LIN {X 0,Y 139.748,Z 528.406,A -85,B 0,C 180,E1 -25612.878,E2 -25612.878} C_VEL
LIN {X 0,Y 135.039,Z 532.973,A -85,B 0,C 180,E1 -25616.378,E2 -25616.378} C_VEL
LIN {X 0,Y 130.036,Z 537.238,A -85,B 0,C 180,E1 -25620.892,E2 -25620.892} C_VEL
LIN {X 0,Y 125.044,Z 540.854,A -85,B 0,C 180,E1 -25626.83,E2 -25626.83} C_VEL
LIN {X 0,Y 123.078,Z 542.06,A -85,B 0,C 180,E1 -25629.962,E2 -25629.962} C_VEL
LIN {X 0,Y 120.547,Z 543.249,A -85,B 0,C 180,E1 -25636.512,E2 -25636.512} C_VEL
LIN {X 0,Y 119.471,Z 542.937,A -85,B 0,C 180,E1 -25643.241,E2 -25643.241} C_VEL
LIN {X 0,Y 119.487,Z 541.317,A -85,B 0,C 180,E1 -25649.219,E2 -25649.219} C_VEL
LIN {X 0,Y 119.402,Z 538.391,A -85,B 0,C 180,E1 -25655.063,E2 -25655.063} C_VEL
LIN {X 0,Y 119.834,Z 534.742,A -85,B 0,C 180,E1 -25660.131,E2 -25660.131} C_VEL
LIN {X 0,Y 120.849,Z 529.936,A -85,B 0,C 180,E1 -25665.168,E2 -25665.168} C_VEL
LIN {X 0,Y 122.779,Z 523.85,A -85,B 0,C 180,E1 -25670.084,E2 -25670.084} C_VEL
LIN {X 0,Y 125.465,Z 516.248,A -85,B 0,C 180,E1 -25674.839,E2 -25674.839} C_VEL
LIN {X 0,Y 127.649,Z 509.707,A -85,B 0,C 180,E1 -25678.109,E2 -25678.109} C_VEL
LIN {X 0,Y 129.2,Z 505.909,A -85,B 0,C 180,E1 -25679.699,E2 -25679.699} C_VEL
LIN {X 0,Y 130.221,Z 501.642,A -85,B 0,C 180,E1 -25681.43,E2 -25681.43} C_VEL
LIN {X 0,Y 130.169,Z 494.346,A -85,B 0,C 180,E1 -25684.371,E2 -25684.371} C_VEL
LIN {X 0,Y 130.081,Z 486.628,A -85,B 0,C 180,E1 -25687.131,E2 -25687.131} C_VEL
LIN {X 0,Y 130.988,Z 481.594,A -85,B 0,C 180,E1 -25688.495,E2 -25688.495} C_VEL
LIN {X 0,Y 133.452,Z 473.066,A -85,B 0,C 180,E1 -25690.171,E2 -25690.171} C_VEL
LIN {X 0,Y 136.354,Z 460.646,A -85,B 0,C 180,E1 -25692.067,E2 -25692.067} C_VEL
LIN {X 0,Y 138.723,Z 447.504,A -85,B 0,C 180,E1 -25693.398,E2 -25693.398} C_VEL
LIN {X 0,Y 140.113,Z 434.838,A -85,B 0,C 180,E1 -25694.224,E2 -25694.224} C_VEL
LIN {X 0,Y 142.429,Z 397.329,A -85,B 0,C 180,E1 -25695.919,E2 -25695.919} C_VEL
LIN {X 0,Y 141.717,Z 386.256,A -85,B 0,C 180,E1 -25696.887,E2 -25696.887} C_VEL
LIN {X 0,Y 137.465,Z 373.788,A -85,B 0,C 180,E1 -25699.297,E2 -25699.297} C_VEL
LIN {X 0,Y 132.823,Z 362.78,A -85,B 0,C 180,E1 -25702.028,E2 -25702.028} C_VEL
LIN {X 0,Y 127.538,Z 354.274,A -85,B 0,C 180,E1 -25705.197,E2 -25705.197} C_VEL
LIN {X 0,Y 124.389,Z 349.812,A -85,B 0,C 180,E1 -25707.263,E2 -25707.263} C_VEL
LIN {X 0,Y 121.952,Z 346.24,A -85,B 0,C 180,E1 -25709.016,E2 -25709.016} C_VEL
LIN {X 0,Y 119.65,Z 343.536,A -85,B 0,C 180,E1 -25710.739,E2 -25710.739} C_VEL
LIN {X 0,Y 118.548,Z 341.533,A -85,B 0,C 180,E1 -25711.688,E2 -25711.688} C_VEL
LIN {X 0,Y 116.07,Z 339.331,A -85,B 0,C 180,E1 -25713.719,E2 -25713.719} C_VEL
LIN {X 0,Y 114.968,Z 336.772,A -85,B 0,C 180,E1 -25714.875,E2 -25714.875} C_VEL
LIN {X 0,Y 114.899,Z 336.166,A -85,B 0,C 180,E1 -25715.068,E2 -25715.068} C_VEL
LIN {X 0,Y 114.974,Z 336.161,A -85,B 0,C 180,E1 -25718.484,E2 -25718.484} C_VEL
LIN {X 0,Y 115.14,Z 336.126,A -85,B 0,C 180,E1 -25725.868,E2 -25725.868} C_VEL
LIN {X 0,Y 115.38,Z 336.107,A -85,B 0,C 180,E1 -25729.471,E2 -25729.471} C_VEL
LIN {X 0,Y 115.524,Z 336.065,A -85,B 0,C 180,E1 -25736.512,E2 -25736.512} C_VEL
LIN {X 0,Y 115.985,Z 336.035,A -85,B 0,C 180,E1 -25740,E2 -25740} C_VEL
LIN {X 0,Y 115.35,Z 336.07,A -85,B 0,C 180,E1 -25746.999,E2 -25746.999} C_VEL
LIN {X 0,Y 115.242,Z 336.129,A -85,B 0,C 180,E1 -25752.658,E2 -25752.658} C_VEL
LIN {X 0,Y 115.003,Z 336.158,A -85,B 0,C 180,E1 -25757.792,E2 -25757.792} C_VEL
LIN {X 0,Y 114.94,Z 336.162,A -85,B 0,C 180,E1 -25763.492,E2 -25763.492} C_VEL
LIN {X 0,Y 114.857,Z 336.175,A -85,B 0,C 180,E1 -25771.064,E2 -25771.064} C_VEL
LIN {X 0,Y 114.77,Z 336.18,A -85,B 0,C 180,E1 -25777.76,E2 -25777.76} C_VEL
LIN {X 0,Y 114.826,Z 336.337,A -85,B 0,C 180,E1 -25779.563,E2 -25779.563} C_VEL
LIN {X 0,Y 115.753,Z 338.963,A -85,B 0,C 180,E1 -25780.602,E2 -25780.602} C_VEL
LIN {X 0,Y 117.898,Z 341.218,A -85,B 0,C 180,E1 -25782.432,E2 -25782.432} C_VEL
LIN {X 0,Y 118.746,Z 341.779,A -85,B 0,C 180,E1 -25783.08,E2 -25783.08} C_VEL
LIN {X 0,Y 120.61,Z 344.977,A -85,B 0,C 180,E1 -25784.635,E2 -25784.635} C_VEL
LIN {X 0,Y 122.547,Z 347.185,A -85,B 0,C 180,E1 -25786.04,E2 -25786.04} C_VEL
LIN {X 0,Y 125.082,Z 350.706,A -85,B 0,C 180,E1 -25787.81,E2 -25787.81} C_VEL
LIN {X 0,Y 130.98,Z 359.656,A -85,B 0,C 180,E1 -25791.51,E2 -25791.51} C_VEL
LIN {X 0,Y 135.931,Z 368.292,A -85,B 0,C 180,E1 -25794.301,E2 -25794.301} C_VEL
LIN {X 0,Y 140.566,Z 377.554,A -85,B 0,C 180,E1 -25796.725,E2 -25796.725} C_VEL
LIN {X 0,Y 143.321,Z 384.36,A -85,B 0,C 180,E1 -25798.137,E2 -25798.137} C_VEL
LIN {X 0,Y 139.982,Z 431.241,A -85,B 0,C 180,E1 -25800.18,E2 -25800.18} C_VEL
LIN {X 0,Y 138.259,Z 444.693,A -85,B 0,C 180,E1 -25801.285,E2 -25801.285} C_VEL
LIN {X 0,Y 135.688,Z 457.591,A -85,B 0,C 180,E1 -25802.845,E2 -25802.845} C_VEL
LIN {X 0,Y 132.84,Z 469.466,A -85,B 0,C 180,E1 -25804.963,E2 -25804.963} C_VEL
LIN {X 0,Y 129.653,Z 480.844,A -85,B 0,C 180,E1 -25807.704,E2 -25807.704} C_VEL
LIN {X 0,Y 126.054,Z 491.183,A -85,B 0,C 180,E1 -25810.882,E2 -25810.882} C_VEL
LIN {X 0,Y 122.214,Z 501.266,A -85,B 0,C 180,E1 -25815.005,E2 -25815.005} C_VEL
LIN {X 0,Y 118.712,Z 510.135,A -85,B 0,C 180,E1 -25819.772,E2 -25819.772} C_VEL
LIN {X 0,Y 115.976,Z 517.221,A -85,B 0,C 180,E1 -25824.787,E2 -25824.787} C_VEL
LIN {X 0,Y 114.01,Z 522.883,A -85,B 0,C 180,E1 -25830.003,E2 -25830.003} C_VEL
LIN {X 0,Y 112.849,Z 526.966,A -85,B 0,C 180,E1 -25834.827,E2 -25834.827} C_VEL
LIN {X 0,Y 111.978,Z 530.745,A -85,B 0,C 180,E1 -25840.855,E2 -25840.855} C_VEL
LIN {X 0,Y 111.907,Z 532.439,A -85,B 0,C 180,E1 -25844.552,E2 -25844.552} C_VEL
LIN {X 0,Y 112.52,Z 534.256,A -85,B 0,C 180,E1 -25850.461,E2 -25850.461} C_VEL
LIN {X 0,Y 113.757,Z 534.966,A -85,B 0,C 180,E1 -25855.627,E2 -25855.627} C_VEL
LIN {X 0,Y 116.732,Z 534.61,A -85,B 0,C 180,E1 -25862.553,E2 -25862.553} C_VEL
LIN {X 0,Y 118.978,Z 533.699,A -85,B 0,C 180,E1 -25866.209,E2 -25866.209} C_VEL
LIN {X 0,Y 121.486,Z 532.41,A -85,B 0,C 180,E1 -25869.523,E2 -25869.523} C_VEL
LIN {X 0,Y 125.754,Z 529.728,A -85,B 0,C 180,E1 -25874.093,E2 -25874.093} C_VEL
LIN {X 0,Y 131.124,Z 525.728,A -85,B 0,C 180,E1 -25878.625,E2 -25878.625} C_VEL
LIN {X 0,Y 137.011,Z 520.617,A -85,B 0,C 180,E1 -25882.665,E2 -25882.665} C_VEL
LIN {X 0,Y 143.466,Z 514.096,A -85,B 0,C 180,E1 -25886.388,E2 -25886.388} C_VEL
LIN {X 0,Y 150.547,Z 505.857,A -85,B 0,C 180,E1 -25889.73,E2 -25889.73} C_VEL
LIN {X 0,Y 156.825,Z 497.394,A -85,B 0,C 180,E1 -25892.264,E2 -25892.264} C_VEL
LIN {X 0,Y 162.673,Z 488.098,A -85,B 0,C 180,E1 -25894.403,E2 -25894.403} C_VEL
LIN {X 0,Y 168.006,Z 477.877,A -85,B 0,C 180,E1 -25896.218,E2 -25896.218} C_VEL
LIN {X 0,Y 172.799,Z 466.653,A -85,B 0,C 180,E1 -25897.713,E2 -25897.713} C_VEL
LIN {X 0,Y 176.818,Z 454.72,A -85,B 0,C 180,E1 -25898.887,E2 -25898.887} C_VEL
LIN {X 0,Y 180.007,Z 441.516,A -85,B 0,C 180,E1 -25899.83,E2 -25899.83} C_VEL
LIN {X 0,Y 181.953,Z 429.077,A -85,B 0,C 180,E1 -25900.379,E2 -25900.379} C_VEL
LIN {X 0,Y 183.021,Z 417.526,A -85,B 0,C 180,E1 -25900.768,E2 -25900.768} C_VEL
LIN {X 0,Y 179.727,Z 410.839,A -85,B 0,C 180,E1 -25903.603,E2 -25903.603} C_VEL
LIN {X 0,Y 176.506,Z 404.889,A -85,B 0,C 180,E1 -25906.783,E2 -25906.783} C_VEL
LIN {X 0,Y 174.369,Z 401.21,A -85,B 0,C 180,E1 -25909.226,E2 -25909.226} C_VEL
LIN {X 0,Y 172.892,Z 398.642,A -85,B 0,C 180,E1 -25911.166,E2 -25911.166} C_VEL
LIN {X 0,Y 170.702,Z 394.74,A -85,B 0,C 180,E1 -25914.759,E2 -25914.759} C_VEL
LIN {X 0,Y 168.911,Z 391.63,A -85,B 0,C 180,E1 -25918.878,E2 -25918.878} C_VEL
LIN {X 0,Y 168.596,Z 390.672,A -85,B 0,C 180,E1 -25920,E2 -25920} C_VEL
LIN {X 0,Y 167.449,Z 390.036,A -85,B 0,C 180,E1 -25927.233,E2 -25927.233} C_VEL
LIN {X 0,Y 168.55,Z 391.104,A -85,B 0,C 180,E1 -25933.561,E2 -25933.561} C_VEL
LIN {X 0,Y 170.089,Z 394.454,A -85,B 0,C 180,E1 -25937.726,E2 -25937.726} C_VEL
LIN {X 0,Y 171.264,Z 395.995,A -85,B 0,C 180,E1 -25939.856,E2 -25939.856} C_VEL
LIN {X 0,Y 173.653,Z 401.111,A -85,B 0,C 180,E1 -25943.557,E2 -25943.557} C_VEL
LIN {X 0,Y 175.886,Z 406.084,A -85,B 0,C 180,E1 -25946.348,E2 -25946.348} C_VEL
LIN {X 0,Y 178.896,Z 413.432,A -85,B 0,C 180,E1 -25949.584,E2 -25949.584} C_VEL
LIN {X 0,Y 181.73,Z 420.904,A -85,B 0,C 180,E1 -25952.25,E2 -25952.25} C_VEL
LIN {X 0,Y 182.632,Z 423.59,A -85,B 0,C 180,E1 -25953.058,E2 -25953.058} C_VEL
LIN {X 0,Y 180.595,Z 441.612,A -85,B 0,C 180,E1 -25953.634,E2 -25953.634} C_VEL
LIN {X 0,Y 178.032,Z 454.239,A -85,B 0,C 180,E1 -25954.299,E2 -25954.299} C_VEL
LIN {X 0,Y 174.696,Z 465.563,A -85,B 0,C 180,E1 -25955.135,E2 -25955.135} C_VEL
LIN {X 0,Y 170.087,Z 477.416,A -85,B 0,C 180,E1 -25956.316,E2 -25956.316} C_VEL
LIN {X 0,Y 164.689,Z 488.641,A -85,B 0,C 180,E1 -25957.861,E2 -25957.861} C_VEL
LIN {X 0,Y 159.45,Z 497.74,A -85,B 0,C 180,E1 -25959.524,E2 -25959.524} C_VEL
LIN {X 0,Y 153.164,Z 507.117,A -85,B 0,C 180,E1 -25961.784,E2 -25961.784} C_VEL
LIN {X 0,Y 145.967,Z 516.189,A -85,B 0,C 180,E1 -25964.749,E2 -25964.749} C_VEL
LIN {X 0,Y 139.287,Z 523.526,A -85,B 0,C 180,E1 -25968.042,E2 -25968.042} C_VEL
LIN {X 0,Y 132.255,Z 530.304,A -85,B 0,C 180,E1 -25972.328,E2 -25972.328} C_VEL
LIN {X 0,Y 127.018,Z 534.81,A -85,B 0,C 180,E1 -25976.403,E2 -25976.403} C_VEL
LIN {X 0,Y 123.878,Z 537.201,A -85,B 0,C 180,E1 -25979.294,E2 -25979.294} C_VEL
LIN {X 0,Y 118.533,Z 540.744,A -85,B 0,C 180,E1 -25985.476,E2 -25985.476} C_VEL
LIN {X 0,Y 116.411,Z 541.883,A -85,B 0,C 180,E1 -25988.76,E2 -25988.76} C_VEL
LIN {X 0,Y 113.638,Z 543.001,A -85,B 0,C 180,E1 -25995.675,E2 -25995.675} C_VEL
LIN {X 0,Y 112.423,Z 542.605,A -85,B 0,C 180,E1 -26002.815,E2 -26002.815} C_VEL
LIN {X 0,Y 112.336,Z 541.788,A -85,B 0,C 180,E1 -26006.411,E2 -26006.411} C_VEL
LIN {X 0,Y 112.448,Z 540.571,A -85,B 0,C 180,E1 -26009.997,E2 -26009.997} C_VEL
LIN {X 0,Y 112.322,Z 537.896,A -85,B 0,C 180,E1 -26015.383,E2 -26015.383} C_VEL
LIN {X 0,Y 112.808,Z 534.167,A -85,B 0,C 180,E1 -26020.769,E2 -26020.769} C_VEL
LIN {X 0,Y 113.96,Z 529.276,A -85,B 0,C 180,E1 -26026.109,E2 -26026.109} C_VEL
LIN {X 0,Y 116.116,Z 523.102,A -85,B 0,C 180,E1 -26031.291,E2 -26031.291} C_VEL
LIN {X 0,Y 119.034,Z 515.391,A -85,B 0,C 180,E1 -26036.28,E2 -26036.28} C_VEL
LIN {X 0,Y 121.143,Z 509.365,A -85,B 0,C 180,E1 -26039.401,E2 -26039.401} C_VEL
LIN {X 0,Y 124.169,Z 501.883,A -85,B 0,C 180,E1 -26042.524,E2 -26042.524} C_VEL
LIN {X 0,Y 127.226,Z 493.263,A -85,B 0,C 180,E1 -26045.449,E2 -26045.449} C_VEL
LIN {X 0,Y 130.988,Z 481.594,A -85,B 0,C 180,E1 -26048.495,E2 -26048.495} C_VEL
LIN {X 0,Y 132.81,Z 482.641,A -85,B 0,C 180,E1 -26049.896,E2 -26049.896} C_VEL
LIN {X 0,Y 132.81,Z 550.306,A -85,B 0,C 180,E1 -26049.896,E2 -26049.896} C_VEL
LIN {X 0,Y 112.28,Z 550.306,A -85,B 0,C 180,E1 -26012.234,E2 -26012.234} C_VEL
LIN {X 0,Y 112.474,Z 548.306,A -85,B 0,C 180,E1 -26011.219,E2 -26011.219} C_VEL
LIN {X 0,Y 112.474,Z 542.531,A -85,B 0,C 180,E1 -26011.219,E2 -26011.219} C_VEL
LIN {X 0,Y 112.448,Z 540.571,A -85,B 0,C 180,E1 -26009.997,E2 -26009.997} C_VEL
LIN {X 0,Y 111.778,Z 539.247,A -85,B 0,C 180,E1 -26012.914,E2 -26012.914} C_VEL
LIN {X 0,Y 110.234,Z 537.667,A -85,B 0,C 180,E1 -26015.768,E2 -26015.768} C_VEL
LIN {X 0,Y 106.956,Z 533.701,A -85,B 0,C 180,E1 -26021.511,E2 -26021.511} C_VEL
LIN {X 0,Y 106.44,Z 531.242,A -85,B 0,C 180,E1 -26024.43,E2 -26024.43} C_VEL
LIN {X 0,Y 106.591,Z 530.347,A -85,B 0,C 180,E1 -26025.386,E2 -26025.386} C_VEL
LIN {X 0,Y 109.011,Z 523.481,A -85,B 0,C 180,E1 -26031.756,E2 -26031.756} C_VEL
LIN {X 0,Y 112.044,Z 515.913,A -85,B 0,C 180,E1 -26037.046,E2 -26037.046} C_VEL
LIN {X 0,Y 114.579,Z 509.293,A -85,B 0,C 180,E1 -26040.708,E2 -26040.708} C_VEL
LIN {X 0,Y 118.166,Z 500.763,A -85,B 0,C 180,E1 -26044.4,E2 -26044.4} C_VEL
LIN {X 0,Y 121.948,Z 490.799,A -85,B 0,C 180,E1 -26047.755,E2 -26047.755} C_VEL
LIN {X 0,Y 125.592,Z 479.732,A -85,B 0,C 180,E1 -26050.577,E2 -26050.577} C_VEL
LIN {X 0,Y 129.109,Z 467.328,A -85,B 0,C 180,E1 -26052.873,E2 -26052.873} C_VEL
LIN {X 0,Y 131.659,Z 455.809,A -85,B 0,C 180,E1 -26054.422,E2 -26054.422} C_VEL
LIN {X 0,Y 133.704,Z 442.907,A -85,B 0,C 180,E1 -26055.605,E2 -26055.605} C_VEL
LIN {X 0,Y 135.239,Z 426.246,A -85,B 0,C 180,E1 -26056.456,E2 -26056.456} C_VEL
LIN {X 0,Y 136.997,Z 398.059,A -85,B 0,C 180,E1 -26057.77,E2 -26057.77} C_VEL
LIN {X 0,Y 136.479,Z 388.679,A -85,B 0,C 180,E1 -26058.621,E2 -26058.621} C_VEL
LIN {X 0,Y 132.52,Z 376.805,A -85,B 0,C 180,E1 -26061.089,E2 -26061.089} C_VEL
LIN {X 0,Y 128.542,Z 367.126,A -85,B 0,C 180,E1 -26063.638,E2 -26063.638} C_VEL
LIN {X 0,Y 123.671,Z 359.17,A -85,B 0,C 180,E1 -26066.816,E2 -26066.816} C_VEL
LIN {X 0,Y 120.424,Z 354.422,A -85,B 0,C 180,E1 -26069.158,E2 -26069.158} C_VEL
LIN {X 0,Y 118.719,Z 351.939,A -85,B 0,C 180,E1 -26070.492,E2 -26070.492} C_VEL
LIN {X 0,Y 116.153,Z 348.364,A -85,B 0,C 180,E1 -26072.647,E2 -26072.647} C_VEL
LIN {X 0,Y 115.403,Z 347.379,A -85,B 0,C 180,E1 -26073.312,E2 -26073.312} C_VEL
LIN {X 0,Y 113.004,Z 344.653,A -85,B 0,C 180,E1 -26075.533,E2 -26075.533} C_VEL
LIN {X 0,Y 112.136,Z 342.754,A -85,B 0,C 180,E1 -26076.513,E2 -26076.513} C_VEL
LIN {X 0,Y 109.351,Z 340.534,A -85,B 0,C 180,E1 -26079.422,E2 -26079.422} C_VEL
LIN {X 0,Y 108.146,Z 338.142,A -85,B 0,C 180,E1 -26081.039,E2 -26081.039} C_VEL
LIN {X 0,Y 107.916,Z 337.008,A -85,B 0,C 180,E1 -26081.489,E2 -26081.489} C_VEL
LIN {X 0,Y 108.295,Z 336.993,A -85,B 0,C 180,E1 -26088.774,E2 -26088.774} C_VEL
LIN {X 0,Y 108.449,Z 336.942,A -85,B 0,C 180,E1 -26096.285,E2 -26096.285} C_VEL
LIN {X 0,Y 108.934,Z 336.914,A -85,B 0,C 180,E1 -26100,E2 -26100} C_VEL
LIN {X 0,Y 108.29,Z 336.95,A -85,B 0,C 180,E1 -26107.458,E2 -26107.458} C_VEL
LIN {X 0,Y 108.164,Z 337.01,A -85,B 0,C 180,E1 -26112.948,E2 -26112.948} C_VEL
LIN {X 0,Y 107.896,Z 337.045,A -85,B 0,C 180,E1 -26119.007,E2 -26119.007} C_VEL
LIN {X 0,Y 107.853,Z 337.048,A -85,B 0,C 180,E1 -26124.186,E2 -26124.186} C_VEL
LIN {X 0,Y 107.779,Z 337.051,A -85,B 0,C 180,E1 -26132.044,E2 -26132.044} C_VEL
LIN {X 0,Y 107.791,Z 337.079,A -85,B 0,C 180,E1 -26133.001,E2 -26133.001} C_VEL
LIN {X 0,Y 108.532,Z 339.574,A -85,B 0,C 180,E1 -26134.185,E2 -26134.185} C_VEL
LIN {X 0,Y 110.337,Z 341.748,A -85,B 0,C 180,E1 -26136.308,E2 -26136.308} C_VEL
LIN {X 0,Y 112.136,Z 342.983,A -85,B 0,C 180,E1 -26138.119,E2 -26138.119} C_VEL
LIN {X 0,Y 113.99,Z 346.133,A -85,B 0,C 180,E1 -26140.055,E2 -26140.055} C_VEL
LIN {X 0,Y 116.076,Z 348.325,A -85,B 0,C 180,E1 -26141.899,E2 -26141.899} C_VEL
LIN {X 0,Y 118.507,Z 351.77,A -85,B 0,C 180,E1 -26143.957,E2 -26143.957} C_VEL
LIN {X 0,Y 122.71,Z 357.834,A -85,B 0,C 180,E1 -26147.129,E2 -26147.129} C_VEL
LIN {X 0,Y 127.287,Z 364.909,A -85,B 0,C 180,E1 -26150.178,E2 -26150.178} C_VEL
LIN {X 0,Y 132.107,Z 373.666,A -85,B 0,C 180,E1 -26153.097,E2 -26153.097} C_VEL
LIN {X 0,Y 136.401,Z 382.721,A -85,B 0,C 180,E1 -26155.527,E2 -26155.527} C_VEL
LIN {X 0,Y 137.681,Z 385.763,A -85,B 0,C 180,E1 -26156.23,E2 -26156.23} C_VEL
LIN {X 0,Y 137.196,Z 395.421,A -85,B 0,C 180,E1 -26156.722,E2 -26156.722} C_VEL
LIN {X 0,Y 134.337,Z 432.384,A -85,B 0,C 180,E1 -26158.383,E2 -26158.383} C_VEL
LIN {X 0,Y 132.557,Z 445.663,A -85,B 0,C 180,E1 -26159.539,E2 -26159.539} C_VEL
LIN {X 0,Y 129.892,Z 458.101,A -85,B 0,C 180,E1 -26161.084,E2 -26161.084} C_VEL
LIN {X 0,Y 126.9,Z 469.914,A -85,B 0,C 180,E1 -26163.261,E2 -26163.261} C_VEL
LIN {X 0,Y 123.519,Z 481.262,A -85,B 0,C 180,E1 -26166.087,E2 -26166.087} C_VEL
LIN {X 0,Y 119.758,Z 491.562,A -85,B 0,C 180,E1 -26169.386,E2 -26169.386} C_VEL
LIN {X 0,Y 116.017,Z 500.807,A -85,B 0,C 180,E1 -26173.28,E2 -26173.28} C_VEL
LIN {X 0,Y 112.25,Z 509.795,A -85,B 0,C 180,E1 -26178.262,E2 -26178.262} C_VEL
LIN {X 0,Y 109.289,Z 517.025,A -85,B 0,C 180,E1 -26183.541,E2 -26183.541} C_VEL
LIN {X 0,Y 107.457,Z 521.902,A -85,B 0,C 180,E1 -26188.129,E2 -26188.129} C_VEL
LIN {X 0,Y 105.766,Z 527.24,A -85,B 0,C 180,E1 -26194.63,E2 -26194.63} C_VEL
LIN {X 0,Y 104.832,Z 531.272,A -85,B 0,C 180,E1 -26201.605,E2 -26201.605} C_VEL
LIN {X 0,Y 104.865,Z 532.919,A -85,B 0,C 180,E1 -26205.553,E2 -26205.553} C_VEL
LIN {X 0,Y 105.515,Z 534.496,A -85,B 0,C 180,E1 -26211.171,E2 -26211.171} C_VEL
LIN {X 0,Y 107.143,Z 535.263,A -85,B 0,C 180,E1 -26217.336,E2 -26217.336} C_VEL
LIN {X 0,Y 110.164,Z 534.899,A -85,B 0,C 180,E1 -26223.967,E2 -26223.967} C_VEL
LIN {X 0,Y 113.055,Z 533.81,A -85,B 0,C 180,E1 -26228.439,E2 -26228.439} C_VEL
LIN {X 0,Y 118.442,Z 531.011,A -85,B 0,C 180,E1 -26234.598,E2 -26234.598} C_VEL
LIN {X 0,Y 124.371,Z 527.048,A -85,B 0,C 180,E1 -26239.72,E2 -26239.72} C_VEL
LIN {X 0,Y 130.465,Z 522.234,A -85,B 0,C 180,E1 -26243.907,E2 -26243.907} C_VEL
LIN {X 0,Y 137.153,Z 516.07,A -85,B 0,C 180,E1 -26247.728,E2 -26247.728} C_VEL
LIN {X 0,Y 144.434,Z 508.335,A -85,B 0,C 180,E1 -26251.149,E2 -26251.149} C_VEL
LIN {X 0,Y 150.868,Z 500.349,A -85,B 0,C 180,E1 -26253.735,E2 -26253.735} C_VEL
LIN {X 0,Y 157.981,Z 489.84,A -85,B 0,C 180,E1 -26256.246,E2 -26256.246} C_VEL
LIN {X 0,Y 163.765,Z 479.448,A -85,B 0,C 180,E1 -26258.134,E2 -26258.134} C_VEL
LIN {X 0,Y 168.707,Z 468.624,A -85,B 0,C 180,E1 -26259.607,E2 -26259.607} C_VEL
LIN {X 0,Y 172.942,Z 456.896,A -85,B 0,C 180,E1 -26260.775,E2 -26260.775} C_VEL
LIN {X 0,Y 176.438,Z 443.601,A -85,B 0,C 180,E1 -26261.757,E2 -26261.757} C_VEL
LIN {X 0,Y 178.686,Z 430.514,A -85,B 0,C 180,E1 -26262.362,E2 -26262.362} C_VEL
LIN {X 0,Y 179.624,Z 421.086,A -85,B 0,C 180,E1 -26262.683,E2 -26262.683} C_VEL
LIN {X 0,Y 176.362,Z 414.445,A -85,B 0,C 180,E1 -26265.826,E2 -26265.826} C_VEL
LIN {X 0,Y 173.363,Z 408.708,A -85,B 0,C 180,E1 -26269.248,E2 -26269.248} C_VEL
LIN {X 0,Y 171.495,Z 405.334,A -85,B 0,C 180,E1 -26271.797,E2 -26271.797} C_VEL
LIN {X 0,Y 169.432,Z 401.474,A -85,B 0,C 180,E1 -26275.417,E2 -26275.417} C_VEL
LIN {X 0,Y 167.748,Z 398.172,A -85,B 0,C 180,E1 -26279.738,E2 -26279.738} C_VEL
LIN {X 0,Y 167.522,Z 397.584,A -85,B 0,C 180,E1 -26280.601,E2 -26280.601} C_VEL
LIN {X 0,Y 166.614,Z 397.162,A -85,B 0,C 180,E1 -26288.186,E2 -26288.186} C_VEL
LIN {X 0,Y 167.511,Z 398.024,A -85,B 0,C 180,E1 -26293.069,E2 -26293.069} C_VEL
LIN {X 0,Y 169.009,Z 401.381,A -85,B 0,C 180,E1 -26297.378,E2 -26297.378} C_VEL
LIN {X 0,Y 169.972,Z 402.756,A -85,B 0,C 180,E1 -26299.234,E2 -26299.234} C_VEL
LIN {X 0,Y 172.118,Z 407.711,A -85,B 0,C 180,E1 -26302.824,E2 -26302.824} C_VEL
LIN {X 0,Y 174.425,Z 413.222,A -85,B 0,C 180,E1 -26305.883,E2 -26305.883} C_VEL
LIN {X 0,Y 177.479,Z 421.435,A -85,B 0,C 180,E1 -26309.336,E2 -26309.336} C_VEL
LIN {X 0,Y 179.239,Z 426.623,A -85,B 0,C 180,E1 -26311.116,E2 -26311.116} C_VEL
LIN {X 0,Y 177.391,Z 441.802,A -85,B 0,C 180,E1 -26311.609,E2 -26311.609} C_VEL
LIN {X 0,Y 174.597,Z 454.82,A -85,B 0,C 180,E1 -26312.293,E2 -26312.293} C_VEL
LIN {X 0,Y 170.842,Z 466.79,A -85,B 0,C 180,E1 -26313.169,E2 -26313.169} C_VEL
LIN {X 0,Y 166.005,Z 478.585,A -85,B 0,C 180,E1 -26314.354,E2 -26314.354} C_VEL
LIN {X 0,Y 160.443,Z 489.534,A -85,B 0,C 180,E1 -26315.866,E2 -26315.866} C_VEL
LIN {X 0,Y 155.06,Z 498.434,A -85,B 0,C 180,E1 -26317.515,E2 -26317.515} C_VEL
LIN {X 0,Y 148.539,Z 507.598,A -85,B 0,C 180,E1 -26319.747,E2 -26319.747} C_VEL
LIN {X 0,Y 141.079,Z 516.535,A -85,B 0,C 180,E1 -26322.709,E2 -26322.709} C_VEL
LIN {X 0,Y 134.106,Z 523.756,A -85,B 0,C 180,E1 -26326.02,E2 -26326.02} C_VEL
LIN {X 0,Y 128.707,Z 528.661,A -85,B 0,C 180,E1 -26329.059,E2 -26329.059} C_VEL
LIN {X 0,Y 122.463,Z 533.813,A -85,B 0,C 180,E1 -26333.46,E2 -26333.46} C_VEL
LIN {X 0,Y 117.826,Z 537.165,A -85,B 0,C 180,E1 -26337.53,E2 -26337.53} C_VEL
LIN {X 0,Y 114.738,Z 539.1,A -85,B 0,C 180,E1 -26340.655,E2 -26340.655} C_VEL
LIN {X 0,Y 112.099,Z 540.618,A -85,B 0,C 180,E1 -26343.966,E2 -26343.966} C_VEL
LIN {X 0,Y 108.047,Z 542.414,A -85,B 0,C 180,E1 -26351.018,E2 -26351.018} C_VEL
LIN {X 0,Y 105.849,Z 542.713,A -85,B 0,C 180,E1 -26358.508,E2 -26358.508} C_VEL
LIN {X 0,Y 105.36,Z 542.254,A -85,B 0,C 180,E1 -26362.331,E2 -26362.331} C_VEL
LIN {X 0,Y 105.246,Z 541.402,A -85,B 0,C 180,E1 -26366.168,E2 -26366.168} C_VEL
LIN {X 0,Y 105.361,Z 540.151,A -85,B 0,C 180,E1 -26369.997,E2 -26369.997} C_VEL
LIN {X 0,Y 105.244,Z 537.401,A -85,B 0,C 180,E1 -26375.746,E2 -26375.746} C_VEL
LIN {X 0,Y 105.815,Z 533.594,A -85,B 0,C 180,E1 -26381.49,E2 -26381.49} C_VEL
LIN {X 0,Y 106.591,Z 530.347,A -85,B 0,C 180,E1 -26385.386,E2 -26385.386} C_VEL
LIN {X 0,Y 106.842,Z 527.656,A -85,B 0,C 180,E1 -26388.182,E2 -26388.182} C_VEL
LIN {X 0,Y 106.071,Z 522.69,A -85,B 0,C 180,E1 -26392.788,E2 -26392.788} C_VEL
LIN {X 0,Y 105.641,Z 517.186,A -85,B 0,C 180,E1 -26397.269,E2 -26397.269} C_VEL
LIN {X 0,Y 106.395,Z 513.493,A -85,B 0,C 180,E1 -26399.752,E2 -26399.752} C_VEL
LIN {X 0,Y 108.363,Z 508.665,A -85,B 0,C 180,E1 -26402.453,E2 -26402.453} C_VEL
LIN {X 0,Y 111.525,Z 501.632,A -85,B 0,C 180,E1 -26405.652,E2 -26405.652} C_VEL
LIN {X 0,Y 115.468,Z 491.896,A -85,B 0,C 180,E1 -26409.155,E2 -26409.155} C_VEL
LIN {X 0,Y 119.207,Z 481.207,A -85,B 0,C 180,E1 -26412.112,E2 -26412.112} C_VEL
LIN {X 0,Y 121.806,Z 473.035,A -85,B 0,C 180,E1 -26413.815,E2 -26413.815} C_VEL
LIN {X 0,Y 124.996,Z 460.764,A -85,B 0,C 180,E1 -26415.793,E2 -26415.793} C_VEL
LIN {X 0,Y 127.548,Z 448.089,A -85,B 0,C 180,E1 -26417.164,E2 -26417.164} C_VEL
LIN {X 0,Y 129.147,Z 435.331,A -85,B 0,C 180,E1 -26418.057,E2 -26418.057} C_VEL
LIN {X 0,Y 131.72,Z 398.47,A -85,B 0,C 180,E1 -26419.795,E2 -26419.795} C_VEL
LIN {X 0,Y 131.244,Z 390.736,A -85,B 0,C 180,E1 -26420.576,E2 -26420.576} C_VEL
LIN {X 0,Y 127.689,Z 379.75,A -85,B 0,C 180,E1 -26423.018,E2 -26423.018} C_VEL
LIN {X 0,Y 124.131,Z 371.032,A -85,B 0,C 180,E1 -26425.516,E2 -26425.516} C_VEL
LIN {X 0,Y 118.446,Z 361.655,A -85,B 0,C 180,E1 -26429.688,E2 -26429.688} C_VEL
LIN {X 0,Y 115.291,Z 357.178,A -85,B 0,C 180,E1 -26432.302,E2 -26432.302} C_VEL
LIN {X 0,Y 112.703,Z 353.448,A -85,B 0,C 180,E1 -26434.714,E2 -26434.714} C_VEL
LIN {X 0,Y 110.096,Z 350.013,A -85,B 0,C 180,E1 -26437.406,E2 -26437.406} C_VEL
LIN {X 0,Y 109.317,Z 348.812,A -85,B 0,C 180,E1 -26438.305,E2 -26438.305} C_VEL
LIN {X 0,Y 106.806,Z 346.222,A -85,B 0,C 180,E1 -26441.29,E2 -26441.29} C_VEL
LIN {X 0,Y 105.624,Z 343.699,A -85,B 0,C 180,E1 -26443.076,E2 -26443.076} C_VEL
LIN {X 0,Y 103.193,Z 342.076,A -85,B 0,C 180,E1 -26446.635,E2 -26446.635} C_VEL
LIN {X 0,Y 101.462,Z 339.05,A -85,B 0,C 180,E1 -26450.154,E2 -26450.154} C_VEL
LIN {X 0,Y 101.222,Z 337.846,A -85,B 0,C 180,E1 -26451.013,E2 -26451.013} C_VEL
LIN {X 0,Y 101.857,Z 337.795,A -85,B 0,C 180,E1 -26460,E2 -26460} C_VEL
LIN {X 0,Y 101.23,Z 337.831,A -85,B 0,C 180,E1 -26467.982,E2 -26467.982} C_VEL
LIN {X 0,Y 101.093,Z 337.888,A -85,B 0,C 180,E1 -26473.291,E2 -26473.291} C_VEL
LIN {X 0,Y 100.88,Z 338.047,A -85,B 0,C 180,E1 -26483.072,E2 -26483.072} C_VEL
LIN {X 0,Y 101.512,Z 340.341,A -85,B 0,C 180,E1 -26484.858,E2 -26484.858} C_VEL
LIN {X 0,Y 103.55,Z 342.812,A -85,B 0,C 180,E1 -26488.642,E2 -26488.642} C_VEL
LIN {X 0,Y 105.581,Z 343.963,A -85,B 0,C 180,E1 -26491.524,E2 -26491.524} C_VEL
LIN {X 0,Y 107.071,Z 346.904,A -85,B 0,C 180,E1 -26493.708,E2 -26493.708} C_VEL
LIN {X 0,Y 109.754,Z 349.454,A -85,B 0,C 180,E1 -26496.803,E2 -26496.803} C_VEL
LIN {X 0,Y 111.93,Z 352.756,A -85,B 0,C 180,E1 -26499.167,E2 -26499.167} C_VEL
LIN {X 0,Y 113.428,Z 354.516,A -85,B 0,C 180,E1 -26500.595,E2 -26500.595} C_VEL
LIN {X 0,Y 116.973,Z 359.668,A -85,B 0,C 180,E1 -26503.745,E2 -26503.745} C_VEL
LIN {X 0,Y 121.255,Z 366.209,A -85,B 0,C 180,E1 -26507.068,E2 -26507.068} C_VEL
LIN {X 0,Y 126.12,Z 374.655,A -85,B 0,C 180,E1 -26510.415,E2 -26510.415} C_VEL
LIN {X 0,Y 131.022,Z 384.848,A -85,B 0,C 180,E1 -26513.483,E2 -26513.483} C_VEL
LIN {X 0,Y 132.447,Z 388.258,A -85,B 0,C 180,E1 -26514.343,E2 -26514.343} C_VEL
LIN {X 0,Y 128.984,Z 432.357,A -85,B 0,C 180,E1 -26516.355,E2 -26516.355} C_VEL
LIN {X 0,Y 126.99,Z 446.3,A -85,B 0,C 180,E1 -26517.582,E2 -26517.582} C_VEL
LIN {X 0,Y 124.231,Z 458.603,A -85,B 0,C 180,E1 -26519.161,E2 -26519.161} C_VEL
LIN {X 0,Y 121.083,Z 470.363,A -85,B 0,C 180,E1 -26521.393,E2 -26521.393} C_VEL
LIN {X 0,Y 117.494,Z 481.68,A -85,B 0,C 180,E1 -26524.303,E2 -26524.303} C_VEL
LIN {X 0,Y 113.578,Z 491.848,A -85,B 0,C 180,E1 -26527.686,E2 -26527.686} C_VEL
LIN {X 0,Y 109.223,Z 501.984,A -85,B 0,C 180,E1 -26532.206,E2 -26532.206} C_VEL
LIN {X 0,Y 105.291,Z 510.818,A -85,B 0,C 180,E1 -26537.474,E2 -26537.474} C_VEL
LIN {X 0,Y 102.178,Z 517.868,A -85,B 0,C 180,E1 -26543.09,E2 -26543.09} C_VEL
LIN {X 0,Y 100.291,Z 522.676,A -85,B 0,C 180,E1 -26547.995,E2 -26547.995} C_VEL
LIN {X 0,Y 98.682,Z 527.502,A -85,B 0,C 180,E1 -26554.386,E2 -26554.386} C_VEL
LIN {X 0,Y 97.807,Z 530.868,A -85,B 0,C 180,E1 -26560.352,E2 -26560.352} C_VEL
LIN {X 0,Y 97.836,Z 533.395,A -85,B 0,C 180,E1 -26566.702,E2 -26566.702} C_VEL
LIN {X 0,Y 98.529,Z 534.736,A -85,B 0,C 180,E1 -26571.985,E2 -26571.985} C_VEL
LIN {X 0,Y 100.614,Z 535.562,A -85,B 0,C 180,E1 -26579.275,E2 -26579.275} C_VEL
LIN {X 0,Y 103.635,Z 535.192,A -85,B 0,C 180,E1 -26585.532,E2 -26585.532} C_VEL
LIN {X 0,Y 107.343,Z 533.926,A -85,B 0,C 180,E1 -26590.902,E2 -26590.902} C_VEL
LIN {X 0,Y 112.598,Z 531.372,A -85,B 0,C 180,E1 -26596.639,E2 -26596.639} C_VEL
LIN {X 0,Y 117.664,Z 528.296,A -85,B 0,C 180,E1 -26600.943,E2 -26600.943} C_VEL
LIN {X 0,Y 124.655,Z 523.302,A -85,B 0,C 180,E1 -26605.681,E2 -26605.681} C_VEL
LIN {X 0,Y 132.109,Z 516.871,A -85,B 0,C 180,E1 -26609.826,E2 -26609.826} C_VEL
LIN {X 0,Y 139.595,Z 509.363,A -85,B 0,C 180,E1 -26613.207,E2 -26613.207} C_VEL
LIN {X 0,Y 146.386,Z 501.416,A -85,B 0,C 180,E1 -26615.813,E2 -26615.813} C_VEL
LIN {X 0,Y 153.531,Z 491.463,A -85,B 0,C 180,E1 -26618.229,E2 -26618.229} C_VEL
LIN {X 0,Y 159.725,Z 480.965,A -85,B 0,C 180,E1 -26620.141,E2 -26620.141} C_VEL
LIN {X 0,Y 164.813,Z 470.464,A -85,B 0,C 180,E1 -26621.588,E2 -26621.588} C_VEL
LIN {X 0,Y 169.253,Z 459.046,A -85,B 0,C 180,E1 -26622.758,E2 -26622.758} C_VEL
LIN {X 0,Y 172.954,Z 446.065,A -85,B 0,C 180,E1 -26623.727,E2 -26623.727} C_VEL
LIN {X 0,Y 175.375,Z 433.781,A -85,B 0,C 180,E1 -26624.322,E2 -26624.322} C_VEL
LIN {X 0,Y 176.408,Z 424.896,A -85,B 0,C 180,E1 -26624.664,E2 -26624.664} C_VEL
LIN {X 0,Y 173.345,Z 418.352,A -85,B 0,C 180,E1 -26628.026,E2 -26628.026} C_VEL
LIN {X 0,Y 171.129,Z 414.096,A -85,B 0,C 180,E1 -26630.887,E2 -26630.887} C_VEL
LIN {X 0,Y 169.747,Z 411.396,A -85,B 0,C 180,E1 -26633.049,E2 -26633.049} C_VEL
LIN {X 0,Y 168.151,Z 408.176,A -85,B 0,C 180,E1 -26636.155,E2 -26636.155} C_VEL
LIN {X 0,Y 166.657,Z 404.862,A -85,B 0,C 180,E1 -26640.453,E2 -26640.453} C_VEL
LIN {X 0,Y 166.172,Z 404.32,A -85,B 0,C 180,E1 -26642.424,E2 -26642.424} C_VEL
LIN {X 0,Y 165.74,Z 404.194,A -85,B 0,C 180,E1 -26648.229,E2 -26648.229} C_VEL
LIN {X 0,Y 166.523,Z 405.107,A -85,B 0,C 180,E1 -26652.761,E2 -26652.761} C_VEL
LIN {X 0,Y 168.076,Z 408.537,A -85,B 0,C 180,E1 -26657.333,E2 -26657.333} C_VEL
LIN {X 0,Y 168.695,Z 409.559,A -85,B 0,C 180,E1 -26658.6,E2 -26658.6} C_VEL
LIN {X 0,Y 170.61,Z 414.328,A -85,B 0,C 180,E1 -26662.079,E2 -26662.079} C_VEL
LIN {X 0,Y 172.791,Z 420.11,A -85,B 0,C 180,E1 -26665.201,E2 -26665.201} C_VEL
LIN {X 0,Y 175.596,Z 428.284,A -85,B 0,C 180,E1 -26668.596,E2 -26668.596} C_VEL
LIN {X 0,Y 176.04,Z 429.715,A -85,B 0,C 180,E1 -26669.094,E2 -26669.094} C_VEL
LIN {X 0,Y 174.163,Z 443.412,A -85,B 0,C 180,E1 -26669.575,E2 -26669.575} C_VEL
LIN {X 0,Y 170.944,Z 456.902,A -85,B 0,C 180,E1 -26670.301,E2 -26670.301} C_VEL
LIN {X 0,Y 167.213,Z 468.008,A -85,B 0,C 180,E1 -26671.123,E2 -26671.123} C_VEL
LIN {X 0,Y 162.129,Z 479.735,A -85,B 0,C 180,E1 -26672.295,E2 -26672.295} C_VEL
LIN {X 0,Y 155.684,Z 491.515,A -85,B 0,C 180,E1 -26673.951,E2 -26673.951} C_VEL
LIN {X 0,Y 149.478,Z 501.009,A -85,B 0,C 180,E1 -26675.8,E2 -26675.8} C_VEL
LIN {X 0,Y 142.835,Z 509.691,A -85,B 0,C 180,E1 -26678.068,E2 -26678.068} C_VEL
LIN {X 0,Y 135.118,Z 518.177,A -85,B 0,C 180,E1 -26681.042,E2 -26681.042} C_VEL
LIN {X 0,Y 127.923,Z 525.002,A -85,B 0,C 180,E1 -26684.419,E2 -26684.419} C_VEL
LIN {X 0,Y 121.308,Z 530.493,A -85,B 0,C 180,E1 -26688.219,E2 -26688.219} C_VEL
LIN {X 0,Y 115.411,Z 534.827,A -85,B 0,C 180,E1 -26692.483,E2 -26692.483} C_VEL
LIN {X 0,Y 111.88,Z 537.138,A -85,B 0,C 180,E1 -26695.57,E2 -26695.57} C_VEL
LIN {X 0,Y 108.588,Z 539.031,A -85,B 0,C 180,E1 -26698.814,E2 -26698.814} C_VEL
LIN {X 0,Y 103.276,Z 541.525,A -85,B 0,C 180,E1 -26705.899,E2 -26705.899} C_VEL
LIN {X 0,Y 99.873,Z 542.503,A -85,B 0,C 180,E1 -26713.649,E2 -26713.649} C_VEL
LIN {X 0,Y 98.888,Z 542.407,A -85,B 0,C 180,E1 -26717.687,E2 -26717.687} C_VEL
LIN {X 0,Y 98.166,Z 541.016,A -85,B 0,C 180,E1 -26725.892,E2 -26725.892} C_VEL
LIN {X 0,Y 98.276,Z 539.731,A -85,B 0,C 180,E1 -26729.997,E2 -26729.997} C_VEL
LIN {X 0,Y 98.189,Z 536.908,A -85,B 0,C 180,E1 -26736.16,E2 -26736.16} C_VEL
LIN {X 0,Y 98.818,Z 533.018,A -85,B 0,C 180,E1 -26742.316,E2 -26742.316} C_VEL
LIN {X 0,Y 100.297,Z 527.959,A -85,B 0,C 180,E1 -26748.377,E2 -26748.377} C_VEL
LIN {X 0,Y 102.902,Z 521.593,A -85,B 0,C 180,E1 -26754.188,E2 -26754.188} C_VEL
LIN {X 0,Y 106.395,Z 513.493,A -85,B 0,C 180,E1 -26759.752,E2 -26759.752} C_VEL
LIN {X 0,Y 107.278,Z 509.66,A -85,B 0,C 180,E1 -26762.097,E2 -26762.097} C_VEL
LIN {X 0,Y 107.706,Z 502.993,A -85,B 0,C 180,E1 -26765.979,E2 -26765.979} C_VEL
LIN {X 0,Y 108.457,Z 495.806,A -85,B 0,C 180,E1 -26769.556,E2 -26769.556} C_VEL
LIN {X 0,Y 109.787,Z 491.11,A -85,B 0,C 180,E1 -26771.349,E2 -26771.349} C_VEL
LIN {X 0,Y 114.039,Z 479.635,A -85,B 0,C 180,E1 -26774.505,E2 -26774.505} C_VEL
LIN {X 0,Y 117.905,Z 467.339,A -85,B 0,C 180,E1 -26776.898,E2 -26776.898} C_VEL
LIN {X 0,Y 120.747,Z 455.729,A -85,B 0,C 180,E1 -26778.532,E2 -26778.532} C_VEL
LIN {X 0,Y 123.014,Z 442.848,A -85,B 0,C 180,E1 -26779.771,E2 -26779.771} C_VEL
LIN {X 0,Y 124.594,Z 427.681,A -85,B 0,C 180,E1 -26780.585,E2 -26780.585} C_VEL
LIN {X 0,Y 126.611,Z 399.243,A -85,B 0,C 180,E1 -26781.947,E2 -26781.947} C_VEL
LIN {X 0,Y 126.247,Z 393.023,A -85,B 0,C 180,E1 -26782.617,E2 -26782.617} C_VEL
LIN {X 0,Y 122.686,Z 381.895,A -85,B 0,C 180,E1 -26785.327,E2 -26785.327} C_VEL
LIN {X 0,Y 120.011,Z 375.294,A -85,B 0,C 180,E1 -26787.411,E2 -26787.411} C_VEL
LIN {X 0,Y 114.906,Z 366.643,A -85,B 0,C 180,E1 -26791.549,E2 -26791.549} C_VEL
LIN {X 0,Y 112.057,Z 362.485,A -85,B 0,C 180,E1 -26794.159,E2 -26794.159} C_VEL
LIN {X 0,Y 109.885,Z 359.234,A -85,B 0,C 180,E1 -26796.39,E2 -26796.39} C_VEL
LIN {X 0,Y 106.89,Z 355.014,A -85,B 0,C 180,E1 -26799.87,E2 -26799.87} C_VEL
LIN {X 0,Y 104.404,Z 351.962,A -85,B 0,C 180,E1 -26803.187,E2 -26803.187} C_VEL
LIN {X 0,Y 103.497,Z 350.225,A -85,B 0,C 180,E1 -26804.658,E2 -26804.658} C_VEL
LIN {X 0,Y 101.205,Z 348.197,A -85,B 0,C 180,E1 -26808.484,E2 -26808.484} C_VEL
LIN {X 0,Y 99.68,Z 344.941,A -85,B 0,C 180,E1 -26812.171,E2 -26812.171} C_VEL
LIN {X 0,Y 97.268,Z 343.234,A -85,B 0,C 180,E1 -26820,E2 -26820} C_VEL
LIN {X 0,Y 96.639,Z 343.337,A -85,B 0,C 180,E1 -26830.476,E2 -26830.476} C_VEL
LIN {X 0,Y 99.356,Z 345.045,A -85,B 0,C 180,E1 -26841.753,E2 -26841.753} C_VEL
LIN {X 0,Y 100.418,Z 347.736,A -85,B 0,C 180,E1 -26844.636,E2 -26844.636} C_VEL
LIN {X 0,Y 102.83,Z 350.073,A -85,B 0,C 180,E1 -26849.011,E2 -26849.011} C_VEL
LIN {X 0,Y 103.653,Z 350.751,A -85,B 0,C 180,E1 -26850.258,E2 -26850.258} C_VEL
LIN {X 0,Y 105.621,Z 353.988,A -85,B 0,C 180,E1 -26853.192,E2 -26853.192} C_VEL
LIN {X 0,Y 107.553,Z 355.949,A -85,B 0,C 180,E1 -26855.551,E2 -26855.551} C_VEL
LIN {X 0,Y 110.306,Z 359.78,A -85,B 0,C 180,E1 -26858.651,E2 -26858.651} C_VEL
LIN {X 0,Y 114.449,Z 366.148,A -85,B 0,C 180,E1 -26862.674,E2 -26862.674} C_VEL
LIN {X 0,Y 118.824,Z 373.207,A -85,B 0,C 180,E1 -26866.29,E2 -26866.29} C_VEL
LIN {X 0,Y 122.894,Z 380.859,A -85,B 0,C 180,E1 -26869.298,E2 -26869.298} C_VEL
LIN {X 0,Y 126.977,Z 389.88,A -85,B 0,C 180,E1 -26872.077,E2 -26872.077} C_VEL
LIN {X 0,Y 127.27,Z 390.575,A -85,B 0,C 180,E1 -26872.268,E2 -26872.268} C_VEL
LIN {X 0,Y 123.838,Z 431.953,A -85,B 0,C 180,E1 -26874.143,E2 -26874.143} C_VEL
LIN {X 0,Y 121.889,Z 445.292,A -85,B 0,C 180,E1 -26875.296,E2 -26875.296} C_VEL
LIN {X 0,Y 118.992,Z 457.986,A -85,B 0,C 180,E1 -26876.888,E2 -26876.888} C_VEL
LIN {X 0,Y 115.898,Z 469.18,A -85,B 0,C 180,E1 -26878.977,E2 -26878.977} C_VEL
LIN {X 0,Y 112.121,Z 480.751,A -85,B 0,C 180,E1 -26881.961,E2 -26881.961} C_VEL
LIN {X 0,Y 107.824,Z 491.253,A -85,B 0,C 180,E1 -26885.45,E2 -26885.45} C_VEL
LIN {X 0,Y 104.033,Z 499.819,A -85,B 0,C 180,E1 -26889.23,E2 -26889.23} C_VEL
LIN {X 0,Y 100.227,Z 507.727,A -85,B 0,C 180,E1 -26893.714,E2 -26893.714} C_VEL
LIN {X 0,Y 96.564,Z 515.425,A -85,B 0,C 180,E1 -26899.52,E2 -26899.52} C_VEL
LIN {X 0,Y 93.862,Z 521.609,A -85,B 0,C 180,E1 -26905.709,E2 -26905.709} C_VEL
LIN {X 0,Y 92.03,Z 526.428,A -85,B 0,C 180,E1 -26912.037,E2 -26912.037} C_VEL
LIN {X 0,Y 90.835,Z 530.343,A -85,B 0,C 180,E1 -26918.905,E2 -26918.905} C_VEL
LIN {X 0,Y 90.606,Z 532.319,A -85,B 0,C 180,E1 -26923.459,E2 -26923.459} C_VEL
LIN {X 0,Y 90.857,Z 533.832,A -85,B 0,C 180,E1 -26928.027,E2 -26928.027} C_VEL
LIN {X 0,Y 91.566,Z 534.971,A -85,B 0,C 180,E1 -26932.92,E2 -26932.92} C_VEL
LIN {X 0,Y 92.646,Z 535.582,A -85,B 0,C 180,E1 -26937.078,E2 -26937.078} C_VEL
LIN {X 0,Y 94.213,Z 535.852,A -85,B 0,C 180,E1 -26941.482,E2 -26941.482} C_VEL
LIN {X 0,Y 97.244,Z 535.481,A -85,B 0,C 180,E1 -26947.345,E2 -26947.345} C_VEL
LIN {X 0,Y 101.832,Z 534.046,A -85,B 0,C 180,E1 -26953.646,E2 -26953.646} C_VEL
LIN {X 0,Y 106.96,Z 531.716,A -85,B 0,C 180,E1 -26958.923,E2 -26958.923} C_VEL
LIN {X 0,Y 113.131,Z 528.226,A -85,B 0,C 180,E1 -26963.865,E2 -26963.865} C_VEL
LIN {X 0,Y 119.824,Z 523.689,A -85,B 0,C 180,E1 -26968.138,E2 -26968.138} C_VEL
LIN {X 0,Y 127.259,Z 517.671,A -85,B 0,C 180,E1 -26972.085,E2 -26972.085} C_VEL
LIN {X 0,Y 135.784,Z 509.533,A -85,B 0,C 180,E1 -26975.737,E2 -26975.737} C_VEL
LIN {X 0,Y 143.517,Z 500.76,A -85,B 0,C 180,E1 -26978.505,E2 -26978.505} C_VEL
LIN {X 0,Y 150.889,Z 490.637,A -85,B 0,C 180,E1 -26980.817,E2 -26980.817} C_VEL
LIN {X 0,Y 157.374,Z 479.807,A -85,B 0,C 180,E1 -26982.666,E2 -26982.666} C_VEL
LIN {X 0,Y 162.635,Z 468.918,A -85,B 0,C 180,E1 -26984.052,E2 -26984.052} C_VEL
LIN {X 0,Y 167.213,Z 456.832,A -85,B 0,C 180,E1 -26985.176,E2 -26985.176} C_VEL
LIN {X 0,Y 170.861,Z 443.641,A -85,B 0,C 180,E1 -26986.067,E2 -26986.067} C_VEL
LIN {X 0,Y 173.196,Z 430.491,A -85,B 0,C 180,E1 -26986.617,E2 -26986.617} C_VEL
LIN {X 0,Y 173.357,Z 428.769,A -85,B 0,C 180,E1 -26986.715,E2 -26986.715} C_VEL
LIN {X 0,Y 170.756,Z 422.977,A -85,B 0,C 180,E1 -26990.021,E2 -26990.021} C_VEL
LIN {X 0,Y 168.499,Z 418.244,A -85,B 0,C 180,E1 -26993.564,E2 -26993.564} C_VEL
LIN {X 0,Y 167,Z 414.986,A -85,B 0,C 180,E1 -26996.683,E2 -26996.683} C_VEL
LIN {X 0,Y 165.573,Z 411.608,A -85,B 0,C 180,E1 -27001.216,E2 -27001.216} C_VEL
LIN {X 0,Y 164.864,Z 411.246,A -85,B 0,C 180,E1 -27008.273,E2 -27008.273} C_VEL
LIN {X 0,Y 165.549,Z 412.152,A -85,B 0,C 180,E1 -27012.465,E2 -27012.465} C_VEL
LIN {X 0,Y 166.932,Z 415.385,A -85,B 0,C 180,E1 -27016.825,E2 -27016.825} C_VEL
LIN {X 0,Y 167.442,Z 416.315,A -85,B 0,C 180,E1 -27017.953,E2 -27017.953} C_VEL
LIN {X 0,Y 169.095,Z 420.861,A -85,B 0,C 180,E1 -27021.246,E2 -27021.246} C_VEL
LIN {X 0,Y 171.055,Z 426.644,A -85,B 0,C 180,E1 -27024.331,E2 -27024.331} C_VEL
LIN {X 0,Y 173.029,Z 432.897,A -85,B 0,C 180,E1 -27027.006,E2 -27027.006} C_VEL
LIN {X 0,Y 171.28,Z 444.24,A -85,B 0,C 180,E1 -27027.444,E2 -27027.444} C_VEL
LIN {X 0,Y 168.079,Z 457.036,A -85,B 0,C 180,E1 -27028.107,E2 -27028.107} C_VEL
LIN {X 0,Y 163.73,Z 469.395,A -85,B 0,C 180,E1 -27029.002,E2 -27029.002} C_VEL
LIN {X 0,Y 158.474,Z 480.77,A -85,B 0,C 180,E1 -27030.139,E2 -27030.139} C_VEL
LIN {X 0,Y 151.851,Z 492.317,A -85,B 0,C 180,E1 -27031.739,E2 -27031.739} C_VEL
LIN {X 0,Y 145.455,Z 501.631,A -85,B 0,C 180,E1 -27033.54,E2 -27033.54} C_VEL
LIN {X 0,Y 138.59,Z 510.154,A -85,B 0,C 180,E1 -27035.767,E2 -27035.767} C_VEL
LIN {X 0,Y 130.584,Z 518.471,A -85,B 0,C 180,E1 -27038.702,E2 -27038.702} C_VEL
LIN {X 0,Y 123.055,Z 525.196,A -85,B 0,C 180,E1 -27042.056,E2 -27042.056} C_VEL
LIN {X 0,Y 116.102,Z 530.596,A -85,B 0,C 180,E1 -27045.88,E2 -27045.88} C_VEL
LIN {X 0,Y 109.852,Z 534.845,A -85,B 0,C 180,E1 -27050.222,E2 -27050.222} C_VEL
LIN {X 0,Y 106.083,Z 537.116,A -85,B 0,C 180,E1 -27053.395,E2 -27053.395} C_VEL
LIN {X 0,Y 102.566,Z 538.944,A -85,B 0,C 180,E1 -27056.755,E2 -27056.755} C_VEL
LIN {X 0,Y 96.831,Z 541.351,A -85,B 0,C 180,E1 -27064.181,E2 -27064.181} C_VEL
LIN {X 0,Y 93.046,Z 542.246,A -85,B 0,C 180,E1 -27072.411,E2 -27072.411} C_VEL
LIN {X 0,Y 91.286,Z 541.55,A -85,B 0,C 180,E1 -27081.139,E2 -27081.139} C_VEL
LIN {X 0,Y 91.078,Z 540.63,A -85,B 0,C 180,E1 -27085.571,E2 -27085.571} C_VEL
LIN {X 0,Y 91.176,Z 539.309,A -85,B 0,C 180,E1 -27089.997,E2 -27089.997} C_VEL
LIN {X 0,Y 91.115,Z 536.412,A -85,B 0,C 180,E1 -27096.641,E2 -27096.641} C_VEL
LIN {X 0,Y 91.853,Z 532.444,A -85,B 0,C 180,E1 -27103.267,E2 -27103.267} C_VEL
LIN {X 0,Y 93.929,Z 526.291,A -85,B 0,C 180,E1 -27110.815,E2 -27110.815} C_VEL
LIN {X 0,Y 96.991,Z 519.552,A -85,B 0,C 180,E1 -27116.925,E2 -27116.925} C_VEL
LIN {X 0,Y 100.12,Z 512.685,A -85,B 0,C 180,E1 -27121.736,E2 -27121.736} C_VEL
LIN {X 0,Y 102.306,Z 507.912,A -85,B 0,C 180,E1 -27124.478,E2 -27124.478} C_VEL
LIN {X 0,Y 106.184,Z 499.512,A -85,B 0,C 180,E1 -27128.349,E2 -27128.349} C_VEL
LIN {X 0,Y 109.787,Z 491.11,A -85,B 0,C 180,E1 -27131.349,E2 -27131.349} C_VEL
LIN {X 0,Y 111.074,Z 486.322,A -85,B 0,C 180,E1 -27133.023,E2 -27133.023} C_VEL
LIN {X 0,Y 111.775,Z 478.222,A -85,B 0,C 180,E1 -27135.943,E2 -27135.943} C_VEL
LIN {X 0,Y 112.346,Z 469.743,A -85,B 0,C 180,E1 -27138.555,E2 -27138.555} C_VEL
LIN {X 0,Y 113.356,Z 464.363,A -85,B 0,C 180,E1 -27139.691,E2 -27139.691} C_VEL
LIN {X 0,Y 116.428,Z 451.357,A -85,B 0,C 180,E1 -27141.343,E2 -27141.343} C_VEL
LIN {X 0,Y 118.518,Z 438.554,A -85,B 0,C 180,E1 -27142.395,E2 -27142.395} C_VEL
LIN {X 0,Y 121.653,Z 400.025,A -85,B 0,C 180,E1 -27144.281,E2 -27144.281} C_VEL
LIN {X 0,Y 121.404,Z 395.406,A -85,B 0,C 180,E1 -27144.814,E2 -27144.814} C_VEL
LIN {X 0,Y 118.128,Z 384.732,A -85,B 0,C 180,E1 -27147.625,E2 -27147.625} C_VEL
LIN {X 0,Y 116.009,Z 379.545,A -85,B 0,C 180,E1 -27149.453,E2 -27149.453} C_VEL
LIN {X 0,Y 111.26,Z 371.249,A -85,B 0,C 180,E1 -27153.758,E2 -27153.758} C_VEL
LIN {X 0,Y 107.444,Z 365.312,A -85,B 0,C 180,E1 -27157.844,E2 -27157.844} C_VEL
LIN {X 0,Y 104.631,Z 361.213,A -85,B 0,C 180,E1 -27161.41,E2 -27161.41} C_VEL
LIN {X 0,Y 102.162,Z 357.761,A -85,B 0,C 180,E1 -27165.088,E2 -27165.088} C_VEL
LIN {X 0,Y 101.66,Z 356.829,A -85,B 0,C 180,E1 -27165.979,E2 -27165.979} C_VEL
LIN {X 0,Y 99.355,Z 354.344,A -85,B 0,C 180,E1 -27170.345,E2 -27170.345} C_VEL
LIN {X 0,Y 98.242,Z 351.662,A -85,B 0,C 180,E1 -27173.457,E2 -27173.457} C_VEL
LIN {X 0,Y 96.367,Z 350.359,A -85,B 0,C 180,E1 -27180,E2 -27180} C_VEL
LIN {X 0,Y 95.761,Z 350.404,A -85,B 0,C 180,E1 -27190.573,E2 -27190.573} C_VEL
LIN {X 0,Y 97.976,Z 352.002,A -85,B 0,C 180,E1 -27200.606,E2 -27200.606} C_VEL
LIN {X 0,Y 99.344,Z 354.991,A -85,B 0,C 180,E1 -27204.403,E2 -27204.403} C_VEL
LIN {X 0,Y 101.839,Z 357.441,A -85,B 0,C 180,E1 -27209.009,E2 -27209.009} C_VEL
LIN {X 0,Y 104.092,Z 360.908,A -85,B 0,C 180,E1 -27212.53,E2 -27212.53} C_VEL
LIN {X 0,Y 105.445,Z 362.486,A -85,B 0,C 180,E1 -27214.299,E2 -27214.299} C_VEL
LIN {X 0,Y 108.523,Z 367.052,A -85,B 0,C 180,E1 -27218,E2 -27218} C_VEL
LIN {X 0,Y 112.669,Z 373.621,A -85,B 0,C 180,E1 -27222.199,E2 -27222.199} C_VEL
LIN {X 0,Y 117.477,Z 382.295,A -85,B 0,C 180,E1 -27226.35,E2 -27226.35} C_VEL
LIN {X 0,Y 122.136,Z 392.699,A -85,B 0,C 180,E1 -27229.937,E2 -27229.937} C_VEL
LIN {X 0,Y 118.827,Z 431.932,A -85,B 0,C 180,E1 -27231.77,E2 -27231.77} C_VEL
LIN {X 0,Y 116.719,Z 445.745,A -85,B 0,C 180,E1 -27232.981,E2 -27232.981} C_VEL
LIN {X 0,Y 113.672,Z 458.394,A -85,B 0,C 180,E1 -27234.579,E2 -27234.579} C_VEL
LIN {X 0,Y 110.413,Z 469.546,A -85,B 0,C 180,E1 -27236.705,E2 -27236.705} C_VEL
LIN {X 0,Y 106.598,Z 480.618,A -85,B 0,C 180,E1 -27239.621,E2 -27239.621} C_VEL
LIN {X 0,Y 102.075,Z 491.153,A -85,B 0,C 180,E1 -27243.197,E2 -27243.197} C_VEL
LIN {X 0,Y 97.385,Z 500.999,A -85,B 0,C 180,E1 -27247.739,E2 -27247.739} C_VEL
LIN {X 0,Y 92.719,Z 510.092,A -85,B 0,C 180,E1 -27253.49,E2 -27253.49} C_VEL
LIN {X 0,Y 89.008,Z 517.417,A -85,B 0,C 180,E1 -27259.77,E2 -27259.77} C_VEL
LIN {X 0,Y 86.727,Z 522.361,A -85,B 0,C 180,E1 -27265.355,E2 -27265.355} C_VEL
LIN {X 0,Y 84.882,Z 526.897,A -85,B 0,C 180,E1 -27271.908,E2 -27271.908} C_VEL
LIN {X 0,Y 83.646,Z 530.905,A -85,B 0,C 180,E1 -27279.677,E2 -27279.677} C_VEL
LIN {X 0,Y 83.517,Z 532.823,A -85,B 0,C 180,E1 -27284.626,E2 -27284.626} C_VEL
LIN {X 0,Y 84.629,Z 535.205,A -85,B 0,C 180,E1 -27294.006,E2 -27294.006} C_VEL
LIN {X 0,Y 86.133,Z 535.924,A -85,B 0,C 180,E1 -27299.316,E2 -27299.316} C_VEL
LIN {X 0,Y 87.983,Z 536.11,A -85,B 0,C 180,E1 -27304.001,E2 -27304.001} C_VEL
LIN {X 0,Y 90.991,Z 535.766,A -85,B 0,C 180,E1 -27309.431,E2 -27309.431} C_VEL
LIN {X 0,Y 96.578,Z 534.15,A -85,B 0,C 180,E1 -27316.698,E2 -27316.698} C_VEL
LIN {X 0,Y 101.472,Z 532.073,A -85,B 0,C 180,E1 -27321.439,E2 -27321.439} C_VEL
LIN {X 0,Y 108.905,Z 528.137,A -85,B 0,C 180,E1 -27327.031,E2 -27327.031} C_VEL
LIN {X 0,Y 116.424,Z 523.214,A -85,B 0,C 180,E1 -27331.449,E2 -27331.449} C_VEL
LIN {X 0,Y 123.951,Z 517.323,A -85,B 0,C 180,E1 -27335.124,E2 -27335.124} C_VEL
LIN {X 0,Y 132.673,Z 509.305,A -85,B 0,C 180,E1 -27338.543,E2 -27338.543} C_VEL
LIN {X 0,Y 139.509,Z 501.835,A -85,B 0,C 180,E1 -27340.837,E2 -27340.837} C_VEL
LIN {X 0,Y 146.957,Z 492.173,A -85,B 0,C 180,E1 -27343.037,E2 -27343.037} C_VEL
LIN {X 0,Y 153.792,Z 481.317,A -85,B 0,C 180,E1 -27344.882,E2 -27344.882} C_VEL
LIN {X 0,Y 159.211,Z 470.784,A -85,B 0,C 180,E1 -27346.206,E2 -27346.206} C_VEL
LIN {X 0,Y 163.909,Z 459.286,A -85,B 0,C 180,E1 -27347.286,E2 -27347.286} C_VEL
LIN {X 0,Y 167.84,Z 446.119,A -85,B 0,C 180,E1 -27348.186,E2 -27348.186} C_VEL
LIN {X 0,Y 170.502,Z 432.818,A -85,B 0,C 180,E1 -27348.784,E2 -27348.784} C_VEL
LIN {X 0,Y 168.312,Z 427.505,A -85,B 0,C 180,E1 -27352.2,E2 -27352.2} C_VEL
LIN {X 0,Y 166.795,Z 424.113,A -85,B 0,C 180,E1 -27355.014,E2 -27355.014} C_VEL
LIN {X 0,Y 165.715,Z 421.615,A -85,B 0,C 180,E1 -27357.569,E2 -27357.569} C_VEL
LIN {X 0,Y 164.535,Z 418.545,A -85,B 0,C 180,E1 -27361.836,E2 -27361.836} C_VEL
LIN {X 0,Y 163.988,Z 418.297,A -85,B 0,C 180,E1 -27368.318,E2 -27368.318} C_VEL
LIN {X 0,Y 164.541,Z 419.056,A -85,B 0,C 180,E1 -27371.963,E2 -27371.963} C_VEL
LIN {X 0,Y 166.175,Z 423.024,A -85,B 0,C 180,E1 -27377.22,E2 -27377.22} C_VEL
LIN {X 0,Y 167.626,Z 427.358,A -85,B 0,C 180,E1 -27380.397,E2 -27380.397} C_VEL
LIN {X 0,Y 169.425,Z 433.433,A -85,B 0,C 180,E1 -27383.613,E2 -27383.613} C_VEL
LIN {X 0,Y 170.19,Z 436.364,A -85,B 0,C 180,E1 -27384.878,E2 -27384.878} C_VEL
LIN {X 0,Y 167.591,Z 449.539,A -85,B 0,C 180,E1 -27385.427,E2 -27385.427} C_VEL
LIN {X 0,Y 163.518,Z 462.973,A -85,B 0,C 180,E1 -27386.204,E2 -27386.204} C_VEL
LIN {X 0,Y 158.888,Z 474.223,A -85,B 0,C 180,E1 -27387.102,E2 -27387.102} C_VEL
LIN {X 0,Y 152.791,Z 485.848,A -85,B 0,C 180,E1 -27388.391,E2 -27388.391} C_VEL
LIN {X 0,Y 146.018,Z 496.322,A -85,B 0,C 180,E1 -27389.959,E2 -27389.959} C_VEL
LIN {X 0,Y 138.813,Z 505.762,A -85,B 0,C 180,E1 -27391.998,E2 -27391.998} C_VEL
LIN {X 0,Y 130.386,Z 514.884,A -85,B 0,C 180,E1 -27394.712,E2 -27394.712} C_VEL
LIN {X 0,Y 122.301,Z 522.256,A -85,B 0,C 180,E1 -27397.799,E2 -27397.799} C_VEL
LIN {X 0,Y 113.471,Z 529.08,A -85,B 0,C 180,E1 -27401.989,E2 -27401.989} C_VEL
LIN {X 0,Y 106.638,Z 533.611,A -85,B 0,C 180,E1 -27406.208,E2 -27406.208} C_VEL
LIN {X 0,Y 100.457,Z 537.087,A -85,B 0,C 180,E1 -27410.973,E2 -27410.973} C_VEL
LIN {X 0,Y 96.696,Z 538.844,A -85,B 0,C 180,E1 -27414.444,E2 -27414.444} C_VEL
LIN {X 0,Y 90.49,Z 541.177,A -85,B 0,C 180,E1 -27422.222,E2 -27422.222} C_VEL
LIN {X 0,Y 88.071,Z 541.776,A -85,B 0,C 180,E1 -27426.481,E2 -27426.481} C_VEL
LIN {X 0,Y 85.009,Z 541.766,A -85,B 0,C 180,E1 -27435.636,E2 -27435.636} C_VEL
LIN {X 0,Y 84.019,Z 540.238,A -85,B 0,C 180,E1 -27445.198,E2 -27445.198} C_VEL
LIN {X 0,Y 84.088,Z 538.858,A -85,B 0,C 180,E1 -27449.997,E2 -27449.997} C_VEL
LIN {X 0,Y 84.07,Z 535.896,A -85,B 0,C 180,E1 -27457.2,E2 -27457.2} C_VEL
LIN {X 0,Y 84.928,Z 531.842,A -85,B 0,C 180,E1 -27464.371,E2 -27464.371} C_VEL
LIN {X 0,Y 87.297,Z 525.564,A -85,B 0,C 180,E1 -27472.479,E2 -27472.479} C_VEL
LIN {X 0,Y 90.658,Z 518.717,A -85,B 0,C 180,E1 -27478.977,E2 -27478.977} C_VEL
LIN {X 0,Y 93.875,Z 512.094,A -85,B 0,C 180,E1 -27483.809,E2 -27483.809} C_VEL
LIN {X 0,Y 96.463,Z 507.009,A -85,B 0,C 180,E1 -27486.811,E2 -27486.811} C_VEL
LIN {X 0,Y 100.634,Z 498.321,A -85,B 0,C 180,E1 -27490.894,E2 -27490.894} C_VEL
LIN {X 0,Y 104.703,Z 489.206,A -85,B 0,C 180,E1 -27494.134,E2 -27494.134} C_VEL
LIN {X 0,Y 109.097,Z 477.928,A -85,B 0,C 180,E1 -27497.115,E2 -27497.115} C_VEL
LIN {X 0,Y 112.847,Z 466.249,A -85,B 0,C 180,E1 -27499.373,E2 -27499.373} C_VEL
LIN {X 0,Y 113.356,Z 464.363,A -85,B 0,C 180,E1 -27499.691,E2 -27499.691} C_VEL
LIN {X 0,Y 114.244,Z 458.886,A -85,B 0,C 180,E1 -27500.732,E2 -27500.732} C_VEL
LIN {X 0,Y 114.212,Z 449.838,A -85,B 0,C 180,E1 -27502.782,E2 -27502.782} C_VEL
LIN {X 0,Y 113.829,Z 440.59,A -85,B 0,C 180,E1 -27504.568,E2 -27504.568} C_VEL
LIN {X 0,Y 114.099,Z 434.803,A -85,B 0,C 180,E1 -27505.159,E2 -27505.159} C_VEL
LIN {X 0,Y 116.916,Z 400.838,A -85,B 0,C 180,E1 -27506.804,E2 -27506.804} C_VEL
LIN {X 0,Y 116.746,Z 397.803,A -85,B 0,C 180,E1 -27507.194,E2 -27507.194} C_VEL
LIN {X 0,Y 113.892,Z 387.973,A -85,B 0,C 180,E1 -27509.982,E2 -27509.982} C_VEL
LIN {X 0,Y 112.244,Z 383.97,A -85,B 0,C 180,E1 -27511.562,E2 -27511.562} C_VEL
LIN {X 0,Y 107.753,Z 375.691,A -85,B 0,C 180,E1 -27516.168,E2 -27516.168} C_VEL
LIN {X 0,Y 104.763,Z 370.986,A -85,B 0,C 180,E1 -27519.756,E2 -27519.756} C_VEL
LIN {X 0,Y 102.537,Z 367.48,A -85,B 0,C 180,E1 -27522.872,E2 -27522.872} C_VEL
LIN {X 0,Y 100.208,Z 363.926,A -85,B 0,C 180,E1 -27526.736,E2 -27526.736} C_VEL
LIN {X 0,Y 97.457,Z 360.041,A -85,B 0,C 180,E1 -27532.768,E2 -27532.768} C_VEL
LIN {X 0,Y 96.905,Z 358.541,A -85,B 0,C 180,E1 -27534.605,E2 -27534.605} C_VEL
LIN {X 0,Y 95.117,Z 357.298,A -85,B 0,C 180,E1 -27542.117,E2 -27542.117} C_VEL
LIN {X 0,Y 94.885,Z 357.471,A -85,B 0,C 180,E1 -27550.671,E2 -27550.671} C_VEL
LIN {X 0,Y 96.673,Z 358.843,A -85,B 0,C 180,E1 -27559.471,E2 -27559.471} C_VEL
LIN {X 0,Y 98.115,Z 361.915,A -85,B 0,C 180,E1 -27563.764,E2 -27563.764} C_VEL
LIN {X 0,Y 100.204,Z 364.259,A -85,B 0,C 180,E1 -27567.937,E2 -27567.937} C_VEL
LIN {X 0,Y 102.432,Z 367.637,A -85,B 0,C 180,E1 -27571.636,E2 -27571.636} C_VEL
LIN {X 0,Y 103.574,Z 369.286,A -85,B 0,C 180,E1 -27573.273,E2 -27573.273} C_VEL
LIN {X 0,Y 106.135,Z 373.265,A -85,B 0,C 180,E1 -27576.582,E2 -27576.582} C_VEL
LIN {X 0,Y 109.734,Z 379.345,A -85,B 0,C 180,E1 -27580.583,E2 -27580.583} C_VEL
LIN {X 0,Y 113.811,Z 387.094,A -85,B 0,C 180,E1 -27584.474,E2 -27584.474} C_VEL
LIN {X 0,Y 117.367,Z 395.241,A -85,B 0,C 180,E1 -27587.533,E2 -27587.533} C_VEL
LIN {X 0,Y 113.874,Z 433.05,A -85,B 0,C 180,E1 -27589.268,E2 -27589.268} C_VEL
LIN {X 0,Y 111.605,Z 446.865,A -85,B 0,C 180,E1 -27590.517,E2 -27590.517} C_VEL
LIN {X 0,Y 108.555,Z 458.799,A -85,B 0,C 180,E1 -27592.049,E2 -27592.049} C_VEL
LIN {X 0,Y 105.12,Z 469.912,A -85,B 0,C 180,E1 -27594.201,E2 -27594.201} C_VEL
LIN {X 0,Y 101.166,Z 480.766,A -85,B 0,C 180,E1 -27597.122,E2 -27597.122} C_VEL
LIN {X 0,Y 96.689,Z 490.622,A -85,B 0,C 180,E1 -27600.501,E2 -27600.501} C_VEL
LIN {X 0,Y 91.753,Z 500.461,A -85,B 0,C 180,E1 -27605.088,E2 -27605.088} C_VEL
LIN {X 0,Y 86.652,Z 509.716,A -85,B 0,C 180,E1 -27611.073,E2 -27611.073} C_VEL
LIN {X 0,Y 82.559,Z 517.153,A -85,B 0,C 180,E1 -27617.716,E2 -27617.716} C_VEL
LIN {X 0,Y 79.563,Z 523.117,A -85,B 0,C 180,E1 -27624.936,E2 -27624.936} C_VEL
LIN {X 0,Y 77.442,Z 528.234,A -85,B 0,C 180,E1 -27633.359,E2 -27633.359} C_VEL
LIN {X 0,Y 76.495,Z 531.466,A -85,B 0,C 180,E1 -27640.592,E2 -27640.592} C_VEL
LIN {X 0,Y 76.457,Z 533.297,A -85,B 0,C 180,E1 -27646.011,E2 -27646.011} C_VEL
LIN {X 0,Y 77.757,Z 535.446,A -85,B 0,C 180,E1 -27655.332,E2 -27655.332} C_VEL
LIN {X 0,Y 79.757,Z 536.245,A -85,B 0,C 180,E1 -27661.922,E2 -27661.922} C_VEL
LIN {X 0,Y 81.935,Z 536.363,A -85,B 0,C 180,E1 -27666.904,E2 -27666.904} C_VEL
LIN {X 0,Y 84.868,Z 536.053,A -85,B 0,C 180,E1 -27671.815,E2 -27671.815} C_VEL
LIN {X 0,Y 87.943,Z 535.385,A -85,B 0,C 180,E1 -27675.995,E2 -27675.995} C_VEL
LIN {X 0,Y 91.633,Z 534.225,A -85,B 0,C 180,E1 -27680.087,E2 -27680.087} C_VEL
LIN {X 0,Y 96.219,Z 532.424,A -85,B 0,C 180,E1 -27684.244,E2 -27684.244} C_VEL
LIN {X 0,Y 102.606,Z 529.349,A -85,B 0,C 180,E1 -27688.895,E2 -27688.895} C_VEL
LIN {X 0,Y 110.837,Z 524.493,A -85,B 0,C 180,E1 -27693.649,E2 -27693.649} C_VEL
LIN {X 0,Y 119.62,Z 518.125,A -85,B 0,C 180,E1 -27697.727,E2 -27697.727} C_VEL
LIN {X 0,Y 127.497,Z 511.329,A -85,B 0,C 180,E1 -27700.686,E2 -27700.686} C_VEL
LIN {X 0,Y 135.741,Z 502.882,A -85,B 0,C 180,E1 -27703.308,E2 -27703.308} C_VEL
LIN {X 0,Y 143.419,Z 493.454,A -85,B 0,C 180,E1 -27705.428,E2 -27705.428} C_VEL
LIN {X 0,Y 150.456,Z 482.833,A -85,B 0,C 180,E1 -27707.19,E2 -27707.19} C_VEL
LIN {X 0,Y 156.014,Z 472.575,A -85,B 0,C 180,E1 -27708.464,E2 -27708.464} C_VEL
LIN {X 0,Y 161.026,Z 461.011,A -85,B 0,C 180,E1 -27709.533,E2 -27709.533} C_VEL
LIN {X 0,Y 165.107,Z 448.409,A -85,B 0,C 180,E1 -27710.386,E2 -27710.386} C_VEL
LIN {X 0,Y 167.664,Z 436.927,A -85,B 0,C 180,E1 -27710.963,E2 -27710.963} C_VEL
LIN {X 0,Y 165.92,Z 431.844,A -85,B 0,C 180,E1 -27714.683,E2 -27714.683} C_VEL
LIN {X 0,Y 164.577,Z 428.417,A -85,B 0,C 180,E1 -27718.164,E2 -27718.164} C_VEL
LIN {X 0,Y 163.581,Z 425.529,A -85,B 0,C 180,E1 -27722.154,E2 -27722.154} C_VEL
LIN {X 0,Y 163.112,Z 425.351,A -85,B 0,C 180,E1 -27728.363,E2 -27728.363} C_VEL
LIN {X 0,Y 163.571,Z 426.093,A -85,B 0,C 180,E1 -27731.619,E2 -27731.619} C_VEL
LIN {X 0,Y 164.967,Z 429.789,A -85,B 0,C 180,E1 -27736.553,E2 -27736.553} C_VEL
LIN {X 0,Y 165.989,Z 433.405,A -85,B 0,C 180,E1 -27739.236,E2 -27739.236} C_VEL
LIN {X 0,Y 167.132,Z 438.402,A -85,B 0,C 180,E1 -27741.994,E2 -27741.994} C_VEL
LIN {X 0,Y 167.427,Z 440.121,A -85,B 0,C 180,E1 -27742.748,E2 -27742.748} C_VEL
LIN {X 0,Y 164.667,Z 452.155,A -85,B 0,C 180,E1 -27743.231,E2 -27743.231} C_VEL
LIN {X 0,Y 160.554,Z 464.592,A -85,B 0,C 180,E1 -27743.965,E2 -27743.965} C_VEL
LIN {X 0,Y 155.027,Z 476.968,A -85,B 0,C 180,E1 -27744.946,E2 -27744.946} C_VEL
LIN {X 0,Y 148.798,Z 488.038,A -85,B 0,C 180,E1 -27746.178,E2 -27746.178} C_VEL
LIN {X 0,Y 142.622,Z 497.028,A -85,B 0,C 180,E1 -27747.5,E2 -27747.5} C_VEL
LIN {X 0,Y 135.199,Z 506.254,A -85,B 0,C 180,E1 -27749.456,E2 -27749.456} C_VEL
LIN {X 0,Y 126.483,Z 515.237,A -85,B 0,C 180,E1 -27752.071,E2 -27752.071} C_VEL
LIN {X 0,Y 118.083,Z 522.501,A -85,B 0,C 180,E1 -27755.076,E2 -27755.076} C_VEL
LIN {X 0,Y 108.857,Z 529.183,A -85,B 0,C 180,E1 -27759.215,E2 -27759.215} C_VEL
LIN {X 0,Y 101.619,Z 533.63,A -85,B 0,C 180,E1 -27763.429,E2 -27763.429} C_VEL
LIN {X 0,Y 95.031,Z 537.033,A -85,B 0,C 180,E1 -27768.269,E2 -27768.269} C_VEL
LIN {X 0,Y 87.407,Z 540.064,A -85,B 0,C 180,E1 -27775.744,E2 -27775.744} C_VEL
LIN {X 0,Y 81.582,Z 541.543,A -85,B 0,C 180,E1 -27784.482,E2 -27784.482} C_VEL
LIN {X 0,Y 78.135,Z 541.446,A -85,B 0,C 180,E1 -27794.342,E2 -27794.342} C_VEL
LIN {X 0,Y 76.952,Z 539.841,A -85,B 0,C 180,E1 -27804.756,E2 -27804.756} C_VEL
LIN {X 0,Y 76.991,Z 538.389,A -85,B 0,C 180,E1 -27809.996,E2 -27809.996} C_VEL
LIN {X 0,Y 77.011,Z 535.35,A -85,B 0,C 180,E1 -27817.864,E2 -27817.864} C_VEL
LIN {X 0,Y 78.021,Z 531.208,A -85,B 0,C 180,E1 -27825.674,E2 -27825.674} C_VEL
LIN {X 0,Y 80.752,Z 524.836,A -85,B 0,C 180,E1 -27834.414,E2 -27834.414} C_VEL
LIN {X 0,Y 84.442,Z 517.88,A -85,B 0,C 180,E1 -27841.34,E2 -27841.34} C_VEL
LIN {X 0,Y 87.731,Z 511.564,A -85,B 0,C 180,E1 -27846.136,E2 -27846.136} C_VEL
LIN {X 0,Y 92.911,Z 502.137,A -85,B 0,C 180,E1 -27851.437,E2 -27851.437} C_VEL
LIN {X 0,Y 97.51,Z 492.648,A -85,B 0,C 180,E1 -27855.371,E2 -27855.371} C_VEL
LIN {X 0,Y 101.945,Z 482.301,A -85,B 0,C 180,E1 -27858.56,E2 -27858.56} C_VEL
LIN {X 0,Y 105.531,Z 472.787,A -85,B 0,C 180,E1 -27860.726,E2 -27860.726} C_VEL
LIN {X 0,Y 109.21,Z 460.658,A -85,B 0,C 180,E1 -27862.78,E2 -27862.78} C_VEL
LIN {X 0,Y 112.115,Z 448.272,A -85,B 0,C 180,E1 -27864.188,E2 -27864.188} C_VEL
LIN {X 0,Y 114.099,Z 434.803,A -85,B 0,C 180,E1 -27865.159,E2 -27865.159} C_VEL
LIN {X 0,Y 114.229,Z 428.997,A -85,B 0,C 180,E1 -27865.707,E2 -27865.707} C_VEL
LIN {X 0,Y 112.163,Z 410.234,A -85,B 0,C 180,E1 -27868.825,E2 -27868.825} C_VEL
LIN {X 0,Y 112.254,Z 404.412,A -85,B 0,C 180,E1 -27869.359,E2 -27869.359} C_VEL
LIN {X 0,Y 112.332,Z 400.278,A -85,B 0,C 180,E1 -27869.74,E2 -27869.74} C_VEL
LIN {X 0,Y 109.778,Z 391.107,A -85,B 0,C 180,E1 -27872.595,E2 -27872.595} C_VEL
LIN {X 0,Y 107.744,Z 386.573,A -85,B 0,C 180,E1 -27874.786,E2 -27874.786} C_VEL
LIN {X 0,Y 104.387,Z 380.314,A -85,B 0,C 180,E1 -27878.771,E2 -27878.771} C_VEL
LIN {X 0,Y 102.148,Z 376.539,A -85,B 0,C 180,E1 -27881.835,E2 -27881.835} C_VEL
LIN {X 0,Y 100.345,Z 373.569,A -85,B 0,C 180,E1 -27884.656,E2 -27884.656} C_VEL
LIN {X 0,Y 98.079,Z 369.839,A -85,B 0,C 180,E1 -27888.962,E2 -27888.962} C_VEL
LIN {X 0,Y 96.065,Z 366.646,A -85,B 0,C 180,E1 -27894.089,E2 -27894.089} C_VEL
LIN {X 0,Y 95.611,Z 365.405,A -85,B 0,C 180,E1 -27895.785,E2 -27895.785} C_VEL
LIN {X 0,Y 94.232,Z 364.345,A -85,B 0,C 180,E1 -27902.137,E2 -27902.137} C_VEL
LIN {X 0,Y 94.012,Z 364.539,A -85,B 0,C 180,E1 -27910.772,E2 -27910.772} C_VEL
LIN {X 0,Y 95.46,Z 365.883,A -85,B 0,C 180,E1 -27918.543,E2 -27918.543} C_VEL
LIN {X 0,Y 97.216,Z 369.298,A -85,B 0,C 180,E1 -27923.885,E2 -27923.885} C_VEL
LIN {X 0,Y 98.488,Z 370.807,A -85,B 0,C 180,E1 -27926.575,E2 -27926.575} C_VEL
LIN {X 0,Y 101.482,Z 375.551,A -85,B 0,C 180,E1 -27931.801,E2 -27931.801} C_VEL
LIN {X 0,Y 103.9,Z 379.57,A -85,B 0,C 180,E1 -27935.205,E2 -27935.205} C_VEL
LIN {X 0,Y 107.182,Z 385.587,A -85,B 0,C 180,E1 -27939.203,E2 -27939.203} C_VEL
LIN {X 0,Y 110.641,Z 392.635,A -85,B 0,C 180,E1 -27942.833,E2 -27942.833} C_VEL
LIN {X 0,Y 112.732,Z 397.968,A -85,B 0,C 180,E1 -27944.889,E2 -27944.889} C_VEL
LIN {X 0,Y 109.269,Z 433.477,A -85,B 0,C 180,E1 -27946.505,E2 -27946.505} C_VEL
LIN {X 0,Y 106.954,Z 446.886,A -85,B 0,C 180,E1 -27947.708,E2 -27947.708} C_VEL
LIN {X 0,Y 103.67,Z 459.202,A -85,B 0,C 180,E1 -27949.274,E2 -27949.274} C_VEL
LIN {X 0,Y 100.048,Z 470.278,A -85,B 0,C 180,E1 -27951.437,E2 -27951.437} C_VEL
LIN {X 0,Y 95.382,Z 482.063,A -85,B 0,C 180,E1 -27954.667,E2 -27954.667} C_VEL
LIN {X 0,Y 90.476,Z 492.242,A -85,B 0,C 180,E1 -27958.381,E2 -27958.381} C_VEL
LIN {X 0,Y 85.325,Z 501.63,A -85,B 0,C 180,E1 -27963.066,E2 -27963.066} C_VEL
LIN {X 0,Y 79.969,Z 510.703,A -85,B 0,C 180,E1 -27969.423,E2 -27969.423} C_VEL
LIN {X 0,Y 75.613,Z 518.016,A -85,B 0,C 180,E1 -27976.568,E2 -27976.568} C_VEL
LIN {X 0,Y 72.411,Z 523.86,A -85,B 0,C 180,E1 -27984.434,E2 -27984.434} C_VEL
LIN {X 0,Y 70.371,Z 528.488,A -85,B 0,C 180,E1 -27992.909,E2 -27992.909} C_VEL
LIN {X 0,Y 69.349,Z 532.006,A -85,B 0,C 180,E1 -28001.698,E2 -28001.698} C_VEL
LIN {X 0,Y 69.452,Z 533.769,A -85,B 0,C 180,E1 -28007.677,E2 -28007.677} C_VEL
LIN {X 0,Y 70.925,Z 535.685,A -85,B 0,C 180,E1 -28016.897,E2 -28016.897} C_VEL
LIN {X 0,Y 73.575,Z 536.543,A -85,B 0,C 180,E1 -28024.973,E2 -28024.973} C_VEL
LIN {X 0,Y 78.847,Z 536.346,A -85,B 0,C 180,E1 -28034.513,E2 -28034.513} C_VEL
LIN {X 0,Y 82.951,Z 535.523,A -85,B 0,C 180,E1 -28039.691,E2 -28039.691} C_VEL
LIN {X 0,Y 91.254,Z 532.766,A -85,B 0,C 180,E1 -28047.376,E2 -28047.376} C_VEL
LIN {X 0,Y 98.976,Z 529.279,A -85,B 0,C 180,E1 -28052.577,E2 -28052.577} C_VEL
LIN {X 0,Y 107.012,Z 524.753,A -85,B 0,C 180,E1 -28056.85,E2 -28056.85} C_VEL
LIN {X 0,Y 115.545,Z 518.922,A -85,B 0,C 180,E1 -28060.53,E2 -28060.53} C_VEL
LIN {X 0,Y 124.518,Z 511.52,A -85,B 0,C 180,E1 -28063.645,E2 -28063.645} C_VEL
LIN {X 0,Y 133.816,Z 502.256,A -85,B 0,C 180,E1 -28066.322,E2 -28066.322} C_VEL
LIN {X 0,Y 141.252,Z 493.248,A -85,B 0,C 180,E1 -28068.197,E2 -28068.197} C_VEL
LIN {X 0,Y 148.187,Z 483.04,A -85,B 0,C 180,E1 -28069.776,E2 -28069.776} C_VEL
LIN {X 0,Y 153.89,Z 472.785,A -85,B 0,C 180,E1 -28070.972,E2 -28070.972} C_VEL
LIN {X 0,Y 159.194,Z 460.809,A -85,B 0,C 180,E1 -28072.002,E2 -28072.002} C_VEL
LIN {X 0,Y 163.41,Z 447.829,A -85,B 0,C 180,E1 -28072.815,E2 -28072.815} C_VEL
LIN {X 0,Y 164.961,Z 441.215,A -85,B 0,C 180,E1 -28073.21,E2 -28073.21} C_VEL
LIN {X 0,Y 163.968,Z 437.691,A -85,B 0,C 180,E1 -28076.16,E2 -28076.16} C_VEL
LIN {X 0,Y 163.241,Z 435.163,A -85,B 0,C 180,E1 -28078.766,E2 -28078.766} C_VEL
LIN {X 0,Y 162.55,Z 432.473,A -85,B 0,C 180,E1 -28082.478,E2 -28082.478} C_VEL
LIN {X 0,Y 162.192,Z 432.431,A -85,B 0,C 180,E1 -28088.723,E2 -28088.723} C_VEL
LIN {X 0,Y 162.521,Z 433.076,A -85,B 0,C 180,E1 -28091.221,E2 -28091.221} C_VEL
LIN {X 0,Y 163.559,Z 436.343,A -85,B 0,C 180,E1 -28095.738,E2 -28095.738} C_VEL
LIN {X 0,Y 164.408,Z 440.47,A -85,B 0,C 180,E1 -28098.78,E2 -28098.78} C_VEL
LIN {X 0,Y 164.822,Z 443.499,A -85,B 0,C 180,E1 -28100.433,E2 -28100.433} C_VEL
LIN {X 0,Y 161.8,Z 455.126,A -85,B 0,C 180,E1 -28100.981,E2 -28100.981} C_VEL
LIN {X 0,Y 157.015,Z 468.144,A -85,B 0,C 180,E1 -28101.753,E2 -28101.753} C_VEL
LIN {X 0,Y 151.386,Z 479.618,A -85,B 0,C 180,E1 -28102.675,E2 -28102.675} C_VEL
LIN {X 0,Y 144.241,Z 491.217,A -85,B 0,C 180,E1 -28103.993,E2 -28103.993} C_VEL
LIN {X 0,Y 137.999,Z 499.609,A -85,B 0,C 180,E1 -28105.312,E2 -28105.312} C_VEL
LIN {X 0,Y 131.866,Z 506.729,A -85,B 0,C 180,E1 -28106.78,E2 -28106.78} C_VEL
LIN {X 0,Y 122.871,Z 515.588,A -85,B 0,C 180,E1 -28109.273,E2 -28109.273} C_VEL
LIN {X 0,Y 114.156,Z 522.741,A -85,B 0,C 180,E1 -28112.162,E2 -28112.162} C_VEL
LIN {X 0,Y 104.509,Z 529.286,A -85,B 0,C 180,E1 -28116.195,E2 -28116.195} C_VEL
LIN {X 0,Y 96.855,Z 533.648,A -85,B 0,C 180,E1 -28120.364,E2 -28120.364} C_VEL
LIN {X 0,Y 89.834,Z 536.971,A -85,B 0,C 180,E1 -28125.24,E2 -28125.24} C_VEL
LIN {X 0,Y 81.61,Z 539.927,A -85,B 0,C 180,E1 -28132.924,E2 -28132.924} C_VEL
LIN {X 0,Y 78.16,Z 540.821,A -85,B 0,C 180,E1 -28137.346,E2 -28137.346} C_VEL
LIN {X 0,Y 75.209,Z 541.295,A -85,B 0,C 180,E1 -28142.141,E2 -28142.141} C_VEL
LIN {X 0,Y 71.317,Z 541.126,A -85,B 0,C 180,E1 -28152.8,E2 -28152.8} C_VEL
LIN {X 0,Y 70.275,Z 540.479,A -85,B 0,C 180,E1 -28158.458,E2 -28158.458} C_VEL
LIN {X 0,Y 69.878,Z 539.419,A -85,B 0,C 180,E1 -28164.224,E2 -28164.224} C_VEL
LIN {X 0,Y 69.888,Z 537.92,A -85,B 0,C 180,E1 -28169.996,E2 -28169.996} C_VEL
LIN {X 0,Y 69.981,Z 534.801,A -85,B 0,C 180,E1 -28178.66,E2 -28178.66} C_VEL
LIN {X 0,Y 71.174,Z 530.571,A -85,B 0,C 180,E1 -28187.227,E2 -28187.227} C_VEL
LIN {X 0,Y 74.321,Z 524.108,A -85,B 0,C 180,E1 -28196.686,E2 -28196.686} C_VEL
LIN {X 0,Y 78.398,Z 517.022,A -85,B 0,C 180,E1 -28204.07,E2 -28204.07} C_VEL
LIN {X 0,Y 82.813,Z 509.198,A -85,B 0,C 180,E1 -28210.045,E2 -28210.045} C_VEL
LIN {X 0,Y 87.667,Z 500.971,A -85,B 0,C 180,E1 -28214.539,E2 -28214.539} C_VEL
LIN {X 0,Y 92.052,Z 492.49,A -85,B 0,C 180,E1 -28218.101,E2 -28218.101} C_VEL
LIN {X 0,Y 96.74,Z 482.162,A -85,B 0,C 180,E1 -28221.343,E2 -28221.343} C_VEL
LIN {X 0,Y 100.519,Z 472.681,A -85,B 0,C 180,E1 -28223.513,E2 -28223.513} C_VEL
LIN {X 0,Y 104.38,Z 460.595,A -85,B 0,C 180,E1 -28225.562,E2 -28225.562} C_VEL
LIN {X 0,Y 107.582,Z 447.427,A -85,B 0,C 180,E1 -28227.033,E2 -28227.033} C_VEL
LIN {X 0,Y 109.544,Z 434.577,A -85,B 0,C 180,E1 -28227.94,E2 -28227.94} C_VEL
LIN {X 0,Y 112.254,Z 404.412,A -85,B 0,C 180,E1 -28229.359,E2 -28229.359} C_VEL
LIN {X 0,Y 112.096,Z 402.047,A -85,B 0,C 180,E1 -28229.713,E2 -28229.713} C_VEL
LIN {X 0,Y 110.943,Z 399.117,A -85,B 0,C 180,E1 -28230.83,E2 -28230.83} C_VEL
LIN {X 0,Y 109.267,Z 396.925,A -85,B 0,C 180,E1 -28232.313,E2 -28232.313} C_VEL
LIN {X 0,Y 105.159,Z 392.538,A -85,B 0,C 180,E1 -28236.31,E2 -28236.31} C_VEL
LIN {X 0,Y 104.432,Z 391.204,A -85,B 0,C 180,E1 -28237.179,E2 -28237.179} C_VEL
LIN {X 0,Y 101.661,Z 385.678,A -85,B 0,C 180,E1 -28240.928,E2 -28240.928} C_VEL
LIN {X 0,Y 98.676,Z 380.209,A -85,B 0,C 180,E1 -28245.767,E2 -28245.767} C_VEL
LIN {X 0,Y 96.444,Z 376.36,A -85,B 0,C 180,E1 -28250.431,E2 -28250.431} C_VEL
LIN {X 0,Y 94.593,Z 372.836,A -85,B 0,C 180,E1 -28256.006,E2 -28256.006} C_VEL
LIN {X 0,Y 94.413,Z 372.299,A -85,B 0,C 180,E1 -28256.8,E2 -28256.8} C_VEL
LIN {X 0,Y 93.347,Z 371.395,A -85,B 0,C 180,E1 -28262.158,E2 -28262.158} C_VEL
LIN {X 0,Y 93.184,Z 371.646,A -85,B 0,C 180,E1 -28271.363,E2 -28271.363} C_VEL
LIN {X 0,Y 94.242,Z 372.626,A -85,B 0,C 180,E1 -28277.356,E2 -28277.356} C_VEL
LIN {X 0,Y 95.842,Z 376.022,A -85,B 0,C 180,E1 -28282.835,E2 -28282.835} C_VEL
LIN {X 0,Y 96.845,Z 377.377,A -85,B 0,C 180,E1 -28285.199,E2 -28285.199} C_VEL
LIN {X 0,Y 99.466,Z 381.796,A -85,B 0,C 180,E1 -28290.274,E2 -28290.274} C_VEL
LIN {X 0,Y 102.404,Z 387.113,A -85,B 0,C 180,E1 -28294.737,E2 -28294.737} C_VEL
LIN {X 0,Y 106.239,Z 395.078,A -85,B 0,C 180,E1 -28299.593,E2 -28299.593} C_VEL
LIN {X 0,Y 108.328,Z 400.36,A -85,B 0,C 180,E1 -28301.963,E2 -28301.963} C_VEL
LIN {X 0,Y 105.053,Z 433.122,A -85,B 0,C 180,E1 -28303.451,E2 -28303.451} C_VEL
LIN {X 0,Y 102.618,Z 446.726,A -85,B 0,C 180,E1 -28304.629,E2 -28304.629} C_VEL
LIN {X 0,Y 99.382,Z 458.505,A -85,B 0,C 180,E1 -28306.064,E2 -28306.064} C_VEL
LIN {X 0,Y 95.235,Z 470.643,A -85,B 0,C 180,E1 -28308.386,E2 -28308.386} C_VEL
LIN {X 0,Y 90.402,Z 482.15,A -85,B 0,C 180,E1 -28311.547,E2 -28311.547} C_VEL
LIN {X 0,Y 85.072,Z 492.573,A -85,B 0,C 180,E1 -28315.397,E2 -28315.397} C_VEL
LIN {X 0,Y 80.097,Z 501.101,A -85,B 0,C 180,E1 -28319.705,E2 -28319.705} C_VEL
LIN {X 0,Y 74.183,Z 510.332,A -85,B 0,C 180,E1 -28326.261,E2 -28326.261} C_VEL
LIN {X 0,Y 69.363,Z 517.753,A -85,B 0,C 180,E1 -28333.826,E2 -28333.826} C_VEL
LIN {X 0,Y 66.286,Z 522.786,A -85,B 0,C 180,E1 -28340.854,E2 -28340.854} C_VEL
LIN {X 0,Y 63.724,Z 527.688,A -85,B 0,C 180,E1 -28350.005,E2 -28350.005} C_VEL
LIN {X 0,Y 62.359,Z 531.484,A -85,B 0,C 180,E1 -28359.737,E2 -28359.737} C_VEL
LIN {X 0,Y 62.528,Z 534.24,A -85,B 0,C 180,E1 -28369.711,E2 -28369.711} C_VEL
LIN {X 0,Y 64.133,Z 535.919,A -85,B 0,C 180,E1 -28378.755,E2 -28378.755} C_VEL
LIN {X 0,Y 67.625,Z 536.841,A -85,B 0,C 180,E1 -28388.581,E2 -28388.581} C_VEL
LIN {X 0,Y 73.137,Z 536.629,A -85,B 0,C 180,E1 -28397.727,E2 -28397.727} C_VEL
LIN {X 0,Y 78.343,Z 535.642,A -85,B 0,C 180,E1 -28403.845,E2 -28403.845} C_VEL
LIN {X 0,Y 86.559,Z 533.118,A -85,B 0,C 180,E1 -28410.846,E2 -28410.846} C_VEL
LIN {X 0,Y 95.784,Z 529.208,A -85,B 0,C 180,E1 -28416.522,E2 -28416.522} C_VEL
LIN {X 0,Y 104.317,Z 524.571,A -85,B 0,C 180,E1 -28420.602,E2 -28420.602} C_VEL
LIN {X 0,Y 113.299,Z 518.594,A -85,B 0,C 180,E1 -28424.051,E2 -28424.051} C_VEL
LIN {X 0,Y 122.646,Z 511.07,A -85,B 0,C 180,E1 -28426.951,E2 -28426.951} C_VEL
LIN {X 0,Y 130.647,Z 503.346,A -85,B 0,C 180,E1 -28429.041,E2 -28429.041} C_VEL
LIN {X 0,Y 138.3,Z 494.522,A -85,B 0,C 180,E1 -28430.806,E2 -28430.806} C_VEL
LIN {X 0,Y 145.399,Z 484.622,A -85,B 0,C 180,E1 -28432.267,E2 -28432.267} C_VEL
LIN {X 0,Y 152.07,Z 473.028,A -85,B 0,C 180,E1 -28433.543,E2 -28433.543} C_VEL
LIN {X 0,Y 157.117,Z 461.953,A -85,B 0,C 180,E1 -28434.438,E2 -28434.438} C_VEL
LIN {X 0,Y 161.5,Z 449.197,A -85,B 0,C 180,E1 -28435.19,E2 -28435.19} C_VEL
LIN {X 0,Y 162.378,Z 445.826,A -85,B 0,C 180,E1 -28435.394,E2 -28435.394} C_VEL
LIN {X 0,Y 161.586,Z 441.892,A -85,B 0,C 180,E1 -28439.315,E2 -28439.315} C_VEL
LIN {X 0,Y 161.144,Z 439.415,A -85,B 0,C 180,E1 -28443.109,E2 -28443.109} C_VEL
LIN {X 0,Y 160.946,Z 439.434,A -85,B 0,C 180,E1 -28448.791,E2 -28448.791} C_VEL
LIN {X 0,Y 161.18,Z 439.976,A -85,B 0,C 180,E1 -28450.838,E2 -28450.838} C_VEL
LIN {X 0,Y 161.853,Z 443.064,A -85,B 0,C 180,E1 -28455.102,E2 -28455.102} C_VEL
LIN {X 0,Y 162.296,Z 446.454,A -85,B 0,C 180,E1 -28457.645,E2 -28457.645} C_VEL
LIN {X 0,Y 162.325,Z 447.563,A -85,B 0,C 180,E1 -28458.225,E2 -28458.225} C_VEL
LIN {X 0,Y 158.344,Z 460.343,A -85,B 0,C 180,E1 -28458.789,E2 -28458.789} C_VEL
LIN {X 0,Y 152.902,Z 473.105,A -85,B 0,C 180,E1 -28459.562,E2 -28459.562} C_VEL
LIN {X 0,Y 146.366,Z 484.799,A -85,B 0,C 180,E1 -28460.553,E2 -28460.553} C_VEL
LIN {X 0,Y 139.081,Z 495.306,A -85,B 0,C 180,E1 -28461.791,E2 -28461.791} C_VEL
LIN {X 0,Y 131.963,Z 503.894,A -85,B 0,C 180,E1 -28463.261,E2 -28463.261} C_VEL
LIN {X 0,Y 124.192,Z 511.829,A -85,B 0,C 180,E1 -28465.114,E2 -28465.114} C_VEL
LIN {X 0,Y 115.015,Z 519.649,A -85,B 0,C 180,E1 -28467.618,E2 -28467.618} C_VEL
LIN {X 0,Y 106.177,Z 525.921,A -85,B 0,C 180,E1 -28470.625,E2 -28470.625} C_VEL
LIN {X 0,Y 97.719,Z 530.947,A -85,B 0,C 180,E1 -28474.195,E2 -28474.195} C_VEL
LIN {X 0,Y 88.084,Z 535.632,A -85,B 0,C 180,E1 -28479.665,E2 -28479.665} C_VEL
LIN {X 0,Y 80.31,Z 538.545,A -85,B 0,C 180,E1 -28485.562,E2 -28485.562} C_VEL
LIN {X 0,Y 76.043,Z 539.79,A -85,B 0,C 180,E1 -28489.683,E2 -28489.683} C_VEL
LIN {X 0,Y 68.987,Z 541.048,A -85,B 0,C 180,E1 -28499.374,E2 -28499.374} C_VEL
LIN {X 0,Y 64.54,Z 540.805,A -85,B 0,C 180,E1 -28510.928,E2 -28510.928} C_VEL
LIN {X 0,Y 63.313,Z 540.11,A -85,B 0,C 180,E1 -28517.168,E2 -28517.168} C_VEL
LIN {X 0,Y 62.831,Z 538.989,A -85,B 0,C 180,E1 -28523.573,E2 -28523.573} C_VEL
LIN {X 0,Y 62.814,Z 537.453,A -85,B 0,C 180,E1 -28529.995,E2 -28529.995} C_VEL
LIN {X 0,Y 62.959,Z 534.251,A -85,B 0,C 180,E1 -28539.634,E2 -28539.634} C_VEL
LIN {X 0,Y 64.395,Z 529.935,A -85,B 0,C 180,E1 -28549.107,E2 -28549.107} C_VEL
LIN {X 0,Y 67.365,Z 524.399,A -85,B 0,C 180,E1 -28557.995,E2 -28557.995} C_VEL
LIN {X 0,Y 71.731,Z 517.46,A -85,B 0,C 180,E1 -28566,E2 -28566} C_VEL
LIN {X 0,Y 75.22,Z 511.846,A -85,B 0,C 180,E1 -28570.84,E2 -28570.84} C_VEL
LIN {X 0,Y 78.301,Z 507.062,A -85,B 0,C 180,E1 -28574.106,E2 -28574.106} C_VEL
LIN {X 0,Y 83.232,Z 498.802,A -85,B 0,C 180,E1 -28578.532,E2 -28578.532} C_VEL
LIN {X 0,Y 88.646,Z 488.747,A -85,B 0,C 180,E1 -28582.443,E2 -28582.443} C_VEL
LIN {X 0,Y 93.822,Z 477.564,A -85,B 0,C 180,E1 -28585.479,E2 -28585.479} C_VEL
LIN {X 0,Y 98.15,Z 465.983,A -85,B 0,C 180,E1 -28587.754,E2 -28587.754} C_VEL
LIN {X 0,Y 101.885,Z 452.959,A -85,B 0,C 180,E1 -28589.538,E2 -28589.538} C_VEL
LIN {X 0,Y 104.483,Z 439.996,A -85,B 0,C 180,E1 -28590.633,E2 -28590.633} C_VEL
LIN {X 0,Y 106.567,Z 420.987,A -85,B 0,C 180,E1 -28591.586,E2 -28591.586} C_VEL
LIN {X 0,Y 108.201,Z 402.945,A -85,B 0,C 180,E1 -28592.433,E2 -28592.433} C_VEL
LIN {X 0,Y 106.061,Z 394.722,A -85,B 0,C 180,E1 -28595.208,E2 -28595.208} C_VEL
LIN {X 0,Y 104.432,Z 391.204,A -85,B 0,C 180,E1 -28597.179,E2 -28597.179} C_VEL
LIN {X 0,Y 103.15,Z 388.928,A -85,B 0,C 180,E1 -28598.796,E2 -28598.796} C_VEL
LIN {X 0,Y 100.982,Z 386.546,A -85,B 0,C 180,E1 -28601.582,E2 -28601.582} C_VEL
LIN {X 0,Y 97.419,Z 384.319,A -85,B 0,C 180,E1 -28606.86,E2 -28606.86} C_VEL
LIN {X 0,Y 95.104,Z 382.861,A -85,B 0,C 180,E1 -28611.453,E2 -28611.453} C_VEL
LIN {X 0,Y 94.236,Z 381.841,A -85,B 0,C 180,E1 -28613.789,E2 -28613.789} C_VEL
LIN {X 0,Y 93.247,Z 379.186,A -85,B 0,C 180,E1 -28617.841,E2 -28617.841} C_VEL
LIN {X 0,Y 92.462,Z 378.444,A -85,B 0,C 180,E1 -28622.178,E2 -28622.178} C_VEL
LIN {X 0,Y 92.206,Z 378.565,A -85,B 0,C 180,E1 -28630.124,E2 -28630.124} C_VEL
LIN {X 0,Y 93.113,Z 379.597,A -85,B 0,C 180,E1 -28636.437,E2 -28636.437} C_VEL
LIN {X 0,Y 94.794,Z 383.179,A -85,B 0,C 180,E1 -28642.563,E2 -28642.563} C_VEL
LIN {X 0,Y 95.764,Z 384.986,A -85,B 0,C 180,E1 -28645.04,E2 -28645.04} C_VEL
LIN {X 0,Y 97.634,Z 388.311,A -85,B 0,C 180,E1 -28648.908,E2 -28648.908} C_VEL
LIN {X 0,Y 100.163,Z 393.347,A -85,B 0,C 180,E1 -28653.178,E2 -28653.178} C_VEL
LIN {X 0,Y 103.551,Z 401.089,A -85,B 0,C 180,E1 -28657.938,E2 -28657.938} C_VEL
LIN {X 0,Y 104.263,Z 403.405,A -85,B 0,C 180,E1 -28658.916,E2 -28658.916} C_VEL
LIN {X 0,Y 101.023,Z 433.707,A -85,B 0,C 180,E1 -28660.222,E2 -28660.222} C_VEL
LIN {X 0,Y 98.428,Z 447.335,A -85,B 0,C 180,E1 -28661.37,E2 -28661.37} C_VEL
LIN {X 0,Y 95.085,Z 458.917,A -85,B 0,C 180,E1 -28662.74,E2 -28662.74} C_VEL
LIN {X 0,Y 90.719,Z 471.009,A -85,B 0,C 180,E1 -28665.021,E2 -28665.021} C_VEL
LIN {X 0,Y 85.582,Z 482.5,A -85,B 0,C 180,E1 -28668.152,E2 -28668.152} C_VEL
LIN {X 0,Y 79.927,Z 492.905,A -85,B 0,C 180,E1 -28672.016,E2 -28672.016} C_VEL
LIN {X 0,Y 74.015,Z 502.262,A -85,B 0,C 180,E1 -28676.913,E2 -28676.913} C_VEL
LIN {X 0,Y 67.735,Z 511.32,A -85,B 0,C 180,E1 -28683.84,E2 -28683.84} C_VEL
LIN {X 0,Y 62.55,Z 518.615,A -85,B 0,C 180,E1 -28692.007,E2 -28692.007} C_VEL
LIN {X 0,Y 59.224,Z 523.54,A -85,B 0,C 180,E1 -28699.752,E2 -28699.752} C_VEL
LIN {X 0,Y 56.246,Z 528.963,A -85,B 0,C 180,E1 -28711.573,E2 -28711.573} C_VEL
LIN {X 0,Y 55.134,Z 533.039,A -85,B 0,C 180,E1 -28724.776,E2 -28724.776} C_VEL
LIN {X 0,Y 55.683,Z 534.712,A -85,B 0,C 180,E1 -28732.255,E2 -28732.255} C_VEL
LIN {X 0,Y 57.447,Z 536.157,A -85,B 0,C 180,E1 -28741.088,E2 -28741.088} C_VEL
LIN {X 0,Y 61.994,Z 537.14,A -85,B 0,C 180,E1 -28752.864,E2 -28752.864} C_VEL
LIN {X 0,Y 67.633,Z 536.918,A -85,B 0,C 180,E1 -28761.428,E2 -28761.428} C_VEL
LIN {X 0,Y 74.202,Z 535.763,A -85,B 0,C 180,E1 -28768.483,E2 -28768.483} C_VEL
LIN {X 0,Y 82.26,Z 533.464,A -85,B 0,C 180,E1 -28774.711,E2 -28774.711} C_VEL
LIN {X 0,Y 90.171,Z 530.416,A -85,B 0,C 180,E1 -28779.283,E2 -28779.283} C_VEL
LIN {X 0,Y 99.776,Z 525.68,A -85,B 0,C 180,E1 -28783.635,E2 -28783.635} C_VEL
LIN {X 0,Y 109.905,Z 519.422,A -85,B 0,C 180,E1 -28787.216,E2 -28787.216} C_VEL
LIN {X 0,Y 119.001,Z 512.499,A -85,B 0,C 180,E1 -28789.795,E2 -28789.795} C_VEL
LIN {X 0,Y 127.786,Z 504.435,A -85,B 0,C 180,E1 -28791.888,E2 -28791.888} C_VEL
LIN {X 0,Y 136.826,Z 494.354,A -85,B 0,C 180,E1 -28793.738,E2 -28793.738} C_VEL
LIN {X 0,Y 144.592,Z 483.534,A -85,B 0,C 180,E1 -28795.162,E2 -28795.162} C_VEL
LIN {X 0,Y 150.562,Z 473.27,A -85,B 0,C 180,E1 -28796.174,E2 -28796.174} C_VEL
LIN {X 0,Y 156.277,Z 460.849,A -85,B 0,C 180,E1 -28797.064,E2 -28797.064} C_VEL
LIN {X 0,Y 159.836,Z 450.55,A -85,B 0,C 180,E1 -28797.656,E2 -28797.656} C_VEL
LIN {X 0,Y 159.542,Z 448.244,A -85,B 0,C 180,E1 -28800.315,E2 -28800.315} C_VEL
LIN {X 0,Y 159.432,Z 446.304,A -85,B 0,C 180,E1 -28803.159,E2 -28803.159} C_VEL
LIN {X 0,Y 159.307,Z 446.332,A -85,B 0,C 180,E1 -28808.882,E2 -28808.882} C_VEL
LIN {X 0,Y 159.43,Z 446.947,A -85,B 0,C 180,E1 -28810.637,E2 -28810.637} C_VEL
LIN {X 0,Y 159.836,Z 449.799,A -85,B 0,C 180,E1 -28814.598,E2 -28814.598} C_VEL
LIN {X 0,Y 159.924,Z 451.272,A -85,B 0,C 180,E1 -28815.778,E2 -28815.778} C_VEL
LIN {X 0,Y 158.123,Z 457.079,A -85,B 0,C 180,E1 -28816.107,E2 -28816.107} C_VEL
LIN {X 0,Y 153.193,Z 469.277,A -85,B 0,C 180,E1 -28816.725,E2 -28816.725} C_VEL
LIN {X 0,Y 146.533,Z 481.821,A -85,B 0,C 180,E1 -28817.587,E2 -28817.587} C_VEL
LIN {X 0,Y 139.099,Z 492.867,A -85,B 0,C 180,E1 -28818.671,E2 -28818.671} C_VEL
LIN {X 0,Y 132.577,Z 500.933,A -85,B 0,C 180,E1 -28819.786,E2 -28819.786} C_VEL
LIN {X 0,Y 126.127,Z 507.756,A -85,B 0,C 180,E1 -28821.035,E2 -28821.035} C_VEL
LIN {X 0,Y 116.607,Z 516.307,A -85,B 0,C 180,E1 -28823.196,E2 -28823.196} C_VEL
LIN {X 0,Y 107.29,Z 523.174,A -85,B 0,C 180,E1 -28825.746,E2 -28825.746} C_VEL
LIN {X 0,Y 96.801,Z 529.512,A -85,B 0,C 180,E1 -28829.393,E2 -28829.393} C_VEL
LIN {X 0,Y 88.296,Z 533.694,A -85,B 0,C 180,E1 -28833.301,E2 -28833.301} C_VEL
LIN {X 0,Y 80.347,Z 536.852,A -85,B 0,C 180,E1 -28838.067,E2 -28838.067} C_VEL
LIN {X 0,Y 75.401,Z 538.447,A -85,B 0,C 180,E1 -28841.779,E2 -28841.779} C_VEL
LIN {X 0,Y 70.759,Z 539.635,A -85,B 0,C 180,E1 -28845.947,E2 -28845.947} C_VEL
LIN {X 0,Y 62.963,Z 540.8,A -85,B 0,C 180,E1 -28856.07,E2 -28856.07} C_VEL
LIN {X 0,Y 57.856,Z 540.483,A -85,B 0,C 180,E1 -28868.623,E2 -28868.623} C_VEL
LIN {X 0,Y 55.774,Z 538.558,A -85,B 0,C 180,E1 -28882.756,E2 -28882.756} C_VEL
LIN {X 0,Y 55.711,Z 536.984,A -85,B 0,C 180,E1 -28889.995,E2 -28889.995} C_VEL
LIN {X 0,Y 55.942,Z 533.701,A -85,B 0,C 180,E1 -28900.857,E2 -28900.857} C_VEL
LIN {X 0,Y 57.671,Z 529.296,A -85,B 0,C 180,E1 -28911.438,E2 -28911.438} C_VEL
LIN {X 0,Y 61.16,Z 523.672,A -85,B 0,C 180,E1 -28921.132,E2 -28921.132} C_VEL
LIN {X 0,Y 66.067,Z 516.611,A -85,B 0,C 180,E1 -28929.656,E2 -28929.656} C_VEL
LIN {X 0,Y 71.558,Z 508.513,A -85,B 0,C 180,E1 -28936.435,E2 -28936.435} C_VEL
LIN {X 0,Y 76.87,Z 500.612,A -85,B 0,C 180,E1 -28940.991,E2 -28940.991} C_VEL
LIN {X 0,Y 81.886,Z 492.174,A -85,B 0,C 180,E1 -28944.615,E2 -28944.615} C_VEL
LIN {X 0,Y 87.139,Z 481.886,A -85,B 0,C 180,E1 -28947.863,E2 -28947.863} C_VEL
LIN {X 0,Y 91.323,Z 472.468,A -85,B 0,C 180,E1 -28949.963,E2 -28949.963} C_VEL
LIN {X 0,Y 95.573,Z 460.47,A -85,B 0,C 180,E1 -28951.929,E2 -28951.929} C_VEL
LIN {X 0,Y 98.915,Z 448.102,A -85,B 0,C 180,E1 -28953.27,E2 -28953.27} C_VEL
LIN {X 0,Y 101.155,Z 435.352,A -85,B 0,C 180,E1 -28954.163,E2 -28954.163} C_VEL
LIN {X 0,Y 104.152,Z 404.891,A -85,B 0,C 180,E1 -28955.588,E2 -28955.588} C_VEL
LIN {X 0,Y 102.753,Z 399.22,A -85,B 0,C 180,E1 -28957.704,E2 -28957.704} C_VEL
LIN {X 0,Y 99.895,Z 392.643,A -85,B 0,C 180,E1 -28961.875,E2 -28961.875} C_VEL
LIN {X 0,Y 96.859,Z 386.568,A -85,B 0,C 180,E1 -28967.279,E2 -28967.279} C_VEL
LIN {X 0,Y 94.806,Z 382.785,A -85,B 0,C 180,E1 -28972.129,E2 -28972.129} C_VEL
LIN {X 0,Y 94.236,Z 381.841,A -85,B 0,C 180,E1 -28973.789,E2 -28973.789} C_VEL
LIN {X 0,Y 93.512,Z 381.112,A -85,B 0,C 180,E1 -28976.102,E2 -28976.102} C_VEL
LIN {X 0,Y 92.544,Z 381.266,A -85,B 0,C 180,E1 -28979.702,E2 -28979.702} C_VEL
LIN {X 0,Y 91.52,Z 383.435,A -85,B 0,C 180,E1 -28985.799,E2 -28985.799} C_VEL
LIN {X 0,Y 91.408,Z 385.425,A -85,B 0,C 180,E1 -28990.783,E2 -28990.783} C_VEL
LIN {X 0,Y 91.649,Z 386.037,A -85,B 0,C 180,E1 -28993.31,E2 -28993.31} C_VEL
LIN {X 0,Y 92.028,Z 386.659,A -85,B 0,C 180,E1 -28995.636,E2 -28995.636} C_VEL
LIN {X 0,Y 93.904,Z 390.851,A -85,B 0,C 180,E1 -29002.789,E2 -29002.789} C_VEL
LIN {X 0,Y 95.757,Z 394.601,A -85,B 0,C 180,E1 -29007.268,E2 -29007.268} C_VEL
LIN {X 0,Y 98.026,Z 399.667,A -85,B 0,C 180,E1 -29011.597,E2 -29011.597} C_VEL
LIN {X 0,Y 100.464,Z 405.78,A -85,B 0,C 180,E1 -29015.479,E2 -29015.479} C_VEL
LIN {X 0,Y 97.487,Z 433.255,A -85,B 0,C 180,E1 -29016.653,E2 -29016.653} C_VEL
LIN {X 0,Y 94.942,Z 446.494,A -85,B 0,C 180,E1 -29017.703,E2 -29017.703} C_VEL
LIN {X 0,Y 91.309,Z 458.789,A -85,B 0,C 180,E1 -29019.041,E2 -29019.041} C_VEL
LIN {X 0,Y 86.547,Z 471.373,A -85,B 0,C 180,E1 -29021.317,E2 -29021.317} C_VEL
LIN {X 0,Y 81.099,Z 482.85,A -85,B 0,C 180,E1 -29024.367,E2 -29024.367} C_VEL
LIN {X 0,Y 75.671,Z 492.278,A -85,B 0,C 180,E1 -29027.774,E2 -29027.774} C_VEL
LIN {X 0,Y 69.376,Z 501.742,A -85,B 0,C 180,E1 -29032.574,E2 -29032.574} C_VEL
LIN {X 0,Y 62.441,Z 510.948,A -85,B 0,C 180,E1 -29039.575,E2 -29039.575} C_VEL
LIN {X 0,Y 56.617,Z 518.354,A -85,B 0,C 180,E1 -29048.142,E2 -29048.142} C_VEL
LIN {X 0,Y 52.193,Z 524.293,A -85,B 0,C 180,E1 -29058.353,E2 -29058.353} C_VEL
LIN {X 0,Y 49.199,Z 529.166,A -85,B 0,C 180,E1 -29070.509,E2 -29070.509} C_VEL
LIN {X 0,Y 48.036,Z 532.608,A -85,B 0,C 180,E1 -29082.683,E2 -29082.683} C_VEL
LIN {X 0,Y 48.983,Z 535.182,A -85,B 0,C 180,E1 -29095.502,E2 -29095.502} C_VEL
LIN {X 0,Y 50.881,Z 536.392,A -85,B 0,C 180,E1 -29104.027,E2 -29104.027} C_VEL
LIN {X 0,Y 56.784,Z 537.437,A -85,B 0,C 180,E1 -29117.961,E2 -29117.961} C_VEL
LIN {X 0,Y 62.385,Z 537.216,A -85,B 0,C 180,E1 -29125.717,E2 -29125.717} C_VEL
LIN {X 0,Y 70.594,Z 535.891,A -85,B 0,C 180,E1 -29133.644,E2 -29133.644} C_VEL
LIN {X 0,Y 78.338,Z 533.825,A -85,B 0,C 180,E1 -29138.97,E2 -29138.97} C_VEL
LIN {X 0,Y 87.822,Z 530.363,A -85,B 0,C 180,E1 -29143.813,E2 -29143.813} C_VEL
LIN {X 0,Y 96.904,Z 526.067,A -85,B 0,C 180,E1 -29147.433,E2 -29147.433} C_VEL
LIN {X 0,Y 106.868,Z 520.213,A -85,B 0,C 180,E1 -29150.571,E2 -29150.571} C_VEL
LIN {X 0,Y 116.891,Z 512.91,A -85,B 0,C 180,E1 -29153.093,E2 -29153.093} C_VEL
LIN {X 0,Y 126.96,Z 503.855,A -85,B 0,C 180,E1 -29155.161,E2 -29155.161} C_VEL
LIN {X 0,Y 135.725,Z 494.153,A -85,B 0,C 180,E1 -29156.733,E2 -29156.733} C_VEL
LIN {X 0,Y 143.291,Z 483.781,A -85,B 0,C 180,E1 -29157.944,E2 -29157.944} C_VEL
LIN {X 0,Y 149.331,Z 473.602,A -85,B 0,C 180,E1 -29158.84,E2 -29158.84} C_VEL
LIN {X 0,Y 155.11,Z 461.289,A -85,B 0,C 180,E1 -29159.639,E2 -29159.639} C_VEL
LIN {X 0,Y 157.313,Z 455.382,A -85,B 0,C 180,E1 -29160,E2 -29160} C_VEL
LIN {X 0,Y 157.245,Z 453.697,A -85,B 0,C 180,E1 -29162.562,E2 -29162.562} C_VEL
LIN {X 0,Y 157.174,Z 452.944,A -85,B 0,C 180,E1 -29165.131,E2 -29165.131} C_VEL
LIN {X 0,Y 157.178,Z 452.975,A -85,B 0,C 180,E1 -29167.709,E2 -29167.709} C_VEL
LIN {X 0,Y 157.279,Z 453.889,A -85,B 0,C 180,E1 -29170.552,E2 -29170.552} C_VEL
LIN {X 0,Y 157.442,Z 455.59,A -85,B 0,C 180,E1 -29173.224,E2 -29173.224} C_VEL
LIN {X 0,Y 156.972,Z 457.285,A -85,B 0,C 180,E1 -29173.567,E2 -29173.567} C_VEL
LIN {X 0,Y 152.163,Z 468.948,A -85,B 0,C 180,E1 -29174.081,E2 -29174.081} C_VEL
LIN {X 0,Y 145.404,Z 481.504,A -85,B 0,C 180,E1 -29174.825,E2 -29174.825} C_VEL
LIN {X 0,Y 137.84,Z 492.564,A -85,B 0,C 180,E1 -29175.763,E2 -29175.763} C_VEL
LIN {X 0,Y 130.357,Z 501.527,A -85,B 0,C 180,E1 -29176.865,E2 -29176.865} C_VEL
LIN {X 0,Y 123.765,Z 508.271,A -85,B 0,C 180,E1 -29177.978,E2 -29177.978} C_VEL
LIN {X 0,Y 114.007,Z 516.634,A -85,B 0,C 180,E1 -29179.928,E2 -29179.928} C_VEL
LIN {X 0,Y 104.409,Z 523.394,A -85,B 0,C 180,E1 -29182.245,E2 -29182.245} C_VEL
LIN {X 0,Y 93.522,Z 529.636,A -85,B 0,C 180,E1 -29185.601,E2 -29185.601} C_VEL
LIN {X 0,Y 84.592,Z 533.728,A -85,B 0,C 180,E1 -29189.261,E2 -29189.261} C_VEL
LIN {X 0,Y 76.166,Z 536.802,A -85,B 0,C 180,E1 -29193.85,E2 -29193.85} C_VEL
LIN {X 0,Y 70.853,Z 538.352,A -85,B 0,C 180,E1 -29197.478,E2 -29197.478} C_VEL
LIN {X 0,Y 61.274,Z 540.197,A -85,B 0,C 180,E1 -29206.508,E2 -29206.508} C_VEL
LIN {X 0,Y 53.841,Z 540.543,A -85,B 0,C 180,E1 -29218.519,E2 -29218.519} C_VEL
LIN {X 0,Y 51.297,Z 540.14,A -85,B 0,C 180,E1 -29225.725,E2 -29225.725} C_VEL
LIN {X 0,Y 48.749,Z 538.128,A -85,B 0,C 180,E1 -29241.705,E2 -29241.705} C_VEL
LIN {X 0,Y 48.625,Z 536.516,A -85,B 0,C 180,E1 -29249.994,E2 -29249.994} C_VEL
LIN {X 0,Y 48.969,Z 533.151,A -85,B 0,C 180,E1 -29262.426,E2 -29262.426} C_VEL
LIN {X 0,Y 51.08,Z 528.659,A -85,B 0,C 180,E1 -29274.372,E2 -29274.372} C_VEL
LIN {X 0,Y 55.157,Z 522.94,A -85,B 0,C 180,E1 -29284.979,E2 -29284.979} C_VEL
LIN {X 0,Y 60.733,Z 515.725,A -85,B 0,C 180,E1 -29293.965,E2 -29293.965} C_VEL
LIN {X 0,Y 66.111,Z 508.486,A -85,B 0,C 180,E1 -29300.209,E2 -29300.209} C_VEL
LIN {X 0,Y 71.286,Z 501.415,A -85,B 0,C 180,E1 -29304.417,E2 -29304.417} C_VEL
LIN {X 0,Y 77.277,Z 492.016,A -85,B 0,C 180,E1 -29308.489,E2 -29308.489} C_VEL
LIN {X 0,Y 82.835,Z 481.749,A -85,B 0,C 180,E1 -29311.664,E2 -29311.664} C_VEL
LIN {X 0,Y 87.227,Z 472.362,A -85,B 0,C 180,E1 -29313.675,E2 -29313.675} C_VEL
LIN {X 0,Y 92.056,Z 459.274,A -85,B 0,C 180,E1 -29315.685,E2 -29315.685} C_VEL
LIN {X 0,Y 95.438,Z 446.906,A -85,B 0,C 180,E1 -29316.907,E2 -29316.907} C_VEL
LIN {X 0,Y 97.682,Z 434.021,A -85,B 0,C 180,E1 -29317.731,E2 -29317.731} C_VEL
LIN {X 0,Y 100.475,Z 407.058,A -85,B 0,C 180,E1 -29318.918,E2 -29318.918} C_VEL
LIN {X 0,Y 99.686,Z 403.801,A -85,B 0,C 180,E1 -29320.301,E2 -29320.301} C_VEL
LIN {X 0,Y 97.443,Z 398.182,A -85,B 0,C 180,E1 -29324.068,E2 -29324.068} C_VEL
LIN {X 0,Y 95.01,Z 392.77,A -85,B 0,C 180,E1 -29329.074,E2 -29329.074} C_VEL
LIN {X 0,Y 93.304,Z 389.225,A -85,B 0,C 180,E1 -29333.753,E2 -29333.753} C_VEL
LIN {X 0,Y 92.025,Z 385.977,A -85,B 0,C 180,E1 -29339.351,E2 -29339.351} C_VEL
LIN {X 0,Y 91.357,Z 385.365,A -85,B 0,C 180,E1 -29344.412,E2 -29344.412} C_VEL
LIN {X 0,Y 91.649,Z 386.037,A -85,B 0,C 180,E1 -29353.31,E2 -29353.31} C_VEL
LIN {X 0,Y 92.004,Z 386.912,A -85,B 0,C 180,E1 -29355.672,E2 -29355.672} C_VEL
LIN {X 0,Y 92.563,Z 389.614,A -85,B 0,C 180,E1 -29358.909,E2 -29358.909} C_VEL
LIN {X 0,Y 93.145,Z 393.327,A -85,B 0,C 180,E1 -29361.77,E2 -29361.77} C_VEL
LIN {X 0,Y 95.486,Z 404.729,A -85,B 0,C 180,E1 -29368.985,E2 -29368.985} C_VEL
LIN {X 0,Y 97.008,Z 408.887,A -85,B 0,C 180,E1 -29371.914,E2 -29371.914} C_VEL
LIN {X 0,Y 94.002,Z 434.785,A -85,B 0,C 180,E1 -29372.981,E2 -29372.981} C_VEL
LIN {X 0,Y 91.205,Z 448.082,A -85,B 0,C 180,E1 -29373.982,E2 -29373.982} C_VEL
LIN {X 0,Y 87.684,Z 459.333,A -85,B 0,C 180,E1 -29375.142,E2 -29375.142} C_VEL
LIN {X 0,Y 82.773,Z 471.658,A -85,B 0,C 180,E1 -29377.257,E2 -29377.257} C_VEL
LIN {X 0,Y 77.009,Z 483.135,A -85,B 0,C 180,E1 -29380.161,E2 -29380.161} C_VEL
LIN {X 0,Y 70.812,Z 493.252,A -85,B 0,C 180,E1 -29383.734,E2 -29383.734} C_VEL
LIN {X 0,Y 63.861,Z 502.854,A -85,B 0,C 180,E1 -29388.683,E2 -29388.683} C_VEL
LIN {X 0,Y 56.424,Z 511.904,A -85,B 0,C 180,E1 -29395.916,E2 -29395.916} C_VEL
LIN {X 0,Y 50.065,Z 519.192,A -85,B 0,C 180,E1 -29405.101,E2 -29405.101} C_VEL
LIN {X 0,Y 45.172,Z 525.007,A -85,B 0,C 180,E1 -29416.511,E2 -29416.511} C_VEL
LIN {X 0,Y 42.02,Z 529.605,A -85,B 0,C 180,E1 -29430.007,E2 -29430.007} C_VEL
LIN {X 0,Y 40.954,Z 533.126,A -85,B 0,C 180,E1 -29444.923,E2 -29444.923} C_VEL
LIN {X 0,Y 42.452,Z 535.627,A -85,B 0,C 180,E1 -29459.786,E2 -29459.786} C_VEL
LIN {X 0,Y 44.805,Z 536.729,A -85,B 0,C 180,E1 -29468.869,E2 -29468.869} C_VEL
LIN {X 0,Y 48.049,Z 537.433,A -85,B 0,C 180,E1 -29477.007,E2 -29477.007} C_VEL
LIN {X 0,Y 52.127,Z 537.733,A -85,B 0,C 180,E1 -29484.002,E2 -29484.002} C_VEL
LIN {X 0,Y 57.632,Z 537.508,A -85,B 0,C 180,E1 -29490.804,E2 -29490.804} C_VEL
LIN {X 0,Y 67.618,Z 536.018,A -85,B 0,C 180,E1 -29499.308,E2 -29499.308} C_VEL
LIN {X 0,Y 74.94,Z 534.174,A -85,B 0,C 180,E1 -29503.659,E2 -29503.659} C_VEL
LIN {X 0,Y 86.044,Z 530.31,A -85,B 0,C 180,E1 -29508.577,E2 -29508.577} C_VEL
LIN {X 0,Y 96.097,Z 525.649,A -85,B 0,C 180,E1 -29511.951,E2 -29511.951} C_VEL
LIN {X 0,Y 105.909,Z 519.938,A -85,B 0,C 180,E1 -29514.51,E2 -29514.51} C_VEL
LIN {X 0,Y 116.636,Z 512.147,A -85,B 0,C 180,E1 -29516.776,E2 -29516.776} C_VEL
LIN {X 0,Y 126.552,Z 503.272,A -85,B 0,C 180,E1 -29518.483,E2 -29518.483} C_VEL
LIN {X 0,Y 135.554,Z 493.242,A -85,B 0,C 180,E1 -29519.838,E2 -29519.838} C_VEL
LIN {X 0,Y 143.216,Z 482.693,A -85,B 0,C 180,E1 -29520.892,E2 -29520.892} C_VEL
LIN {X 0,Y 149.808,Z 471.377,A -85,B 0,C 180,E1 -29521.713,E2 -29521.713} C_VEL
LIN {X 0,Y 154.288,Z 461.664,A -85,B 0,C 180,E1 -29522.249,E2 -29522.249} C_VEL
LIN {X 0,Y 154.698,Z 460.605,A -85,B 0,C 180,E1 -29522.392,E2 -29522.392} C_VEL
LIN {X 0,Y 154.741,Z 459.612,A -85,B 0,C 180,E1 -29525.212,E2 -29525.212} C_VEL
LIN {X 0,Y 154.745,Z 459.714,A -85,B 0,C 180,E1 -29527.831,E2 -29527.831} C_VEL
LIN {X 0,Y 154.769,Z 460.652,A -85,B 0,C 180,E1 -29530.465,E2 -29530.465} C_VEL
LIN {X 0,Y 154.158,Z 462.569,A -85,B 0,C 180,E1 -29531.171,E2 -29531.171} C_VEL
LIN {X 0,Y 148.041,Z 475.301,A -85,B 0,C 180,E1 -29531.718,E2 -29531.718} C_VEL
LIN {X 0,Y 141.201,Z 486.433,A -85,B 0,C 180,E1 -29532.36,E2 -29532.36} C_VEL
LIN {X 0,Y 133.539,Z 496.476,A -85,B 0,C 180,E1 -29533.18,E2 -29533.18} C_VEL
LIN {X 0,Y 125.103,Z 505.553,A -85,B 0,C 180,E1 -29534.283,E2 -29534.283} C_VEL
LIN {X 0,Y 115.123,Z 514.414,A -85,B 0,C 180,E1 -29535.944,E2 -29535.944} C_VEL
LIN {X 0,Y 105.192,Z 521.583,A -85,B 0,C 180,E1 -29537.806,E2 -29537.806} C_VEL
LIN {X 0,Y 93.866,Z 528.141,A -85,B 0,C 180,E1 -29540.617,E2 -29540.617} C_VEL
LIN {X 0,Y 84.424,Z 532.512,A -85,B 0,C 180,E1 -29543.686,E2 -29543.686} C_VEL
LIN {X 0,Y 72.448,Z 536.753,A -85,B 0,C 180,E1 -29549.175,E2 -29549.175} C_VEL
LIN {X 0,Y 66.76,Z 538.231,A -85,B 0,C 180,E1 -29552.622,E2 -29552.622} C_VEL
LIN {X 0,Y 56.329,Z 539.99,A -85,B 0,C 180,E1 -29561.523,E2 -29561.523} C_VEL
LIN {X 0,Y 47.899,Z 540.247,A -85,B 0,C 180,E1 -29574.056,E2 -29574.056} C_VEL
LIN {X 0,Y 42.764,Z 538.926,A -85,B 0,C 180,E1 -29590.804,E2 -29590.804} C_VEL
LIN {X 0,Y 41.719,Z 537.691,A -85,B 0,C 180,E1 -29600.295,E2 -29600.295} C_VEL
LIN {X 0,Y 41.532,Z 536.04,A -85,B 0,C 180,E1 -29609.993,E2 -29609.993} C_VEL
LIN {X 0,Y 42.034,Z 532.594,A -85,B 0,C 180,E1 -29624.517,E2 -29624.517} C_VEL
LIN {X 0,Y 44.675,Z 528.011,A -85,B 0,C 180,E1 -29638.153,E2 -29638.153} C_VEL
LIN {X 0,Y 50.467,Z 521.04,A -85,B 0,C 180,E1 -29651.405,E2 -29651.405} C_VEL
LIN {X 0,Y 56.984,Z 513.445,A -85,B 0,C 180,E1 -29660.419,E2 -29660.419} C_VEL
LIN {X 0,Y 61.442,Z 507.888,A -85,B 0,C 180,E1 -29665.004,E2 -29665.004} C_VEL
LIN {X 0,Y 67.358,Z 500.227,A -85,B 0,C 180,E1 -29669.396,E2 -29669.396} C_VEL
LIN {X 0,Y 74.512,Z 489.442,A -85,B 0,C 180,E1 -29673.632,E2 -29673.632} C_VEL
LIN {X 0,Y 80.477,Z 478.699,A -85,B 0,C 180,E1 -29676.474,E2 -29676.474} C_VEL
LIN {X 0,Y 85.856,Z 466.658,A -85,B 0,C 180,E1 -29678.601,E2 -29678.601} C_VEL
LIN {X 0,Y 90.117,Z 454.119,A -85,B 0,C 180,E1 -29680.132,E2 -29680.132} C_VEL
LIN {X 0,Y 93.268,Z 441.108,A -85,B 0,C 180,E1 -29681.126,E2 -29681.126} C_VEL
LIN {X 0,Y 95.455,Z 424.937,A -85,B 0,C 180,E1 -29681.86,E2 -29681.86} C_VEL
LIN {X 0,Y 97.079,Z 409.137,A -85,B 0,C 180,E1 -29682.561,E2 -29682.561} C_VEL
LIN {X 0,Y 95.204,Z 403.811,A -85,B 0,C 180,E1 -29686.253,E2 -29686.253} C_VEL
LIN {X 0,Y 93.172,Z 398.79,A -85,B 0,C 180,E1 -29691.17,E2 -29691.17} C_VEL
LIN {X 0,Y 91.914,Z 395.76,A -85,B 0,C 180,E1 -29695.289,E2 -29695.289} C_VEL
LIN {X 0,Y 90.922,Z 392.788,A -85,B 0,C 180,E1 -29700.579,E2 -29700.579} C_VEL
LIN {X 0,Y 90.474,Z 392.409,A -85,B 0,C 180,E1 -29704.455,E2 -29704.455} C_VEL
LIN {X 0,Y 90.716,Z 393.057,A -85,B 0,C 180,E1 -29712.967,E2 -29712.967} C_VEL
LIN {X 0,Y 91.046,Z 393.997,A -85,B 0,C 180,E1 -29715.379,E2 -29715.379} C_VEL
LIN {X 0,Y 92.443,Z 397.41,A -85,B 0,C 180,E1 -29721.332,E2 -29721.332} C_VEL
LIN {X 0,Y 94.015,Z 401.019,A -85,B 0,C 180,E1 -29725.697,E2 -29725.697} C_VEL
LIN {X 0,Y 95.486,Z 404.729,A -85,B 0,C 180,E1 -29728.985,E2 -29728.985} C_VEL
LIN {X 0,Y 95.786,Z 406.969,A -85,B 0,C 180,E1 -29729.879,E2 -29729.879} C_VEL
LIN {X 0,Y 95.553,Z 410.391,A -85,B 0,C 180,E1 -29730.208,E2 -29730.208} C_VEL
LIN {X 0,Y 94.849,Z 414.259,A -85,B 0,C 180,E1 -29729.945,E2 -29729.945} C_VEL
LIN {X 0,Y 92.758,Z 423.587,A -85,B 0,C 180,E1 -29728.667,E2 -29728.667} C_VEL
LIN {X 0,Y 92.445,Z 425.803,A -85,B 0,C 180,E1 -29728.64,E2 -29728.64} C_VEL
LIN {X 0,Y 90.474,Z 438.907,A -85,B 0,C 180,E1 -29729.193,E2 -29729.193} C_VEL
LIN {X 0,Y 87.429,Z 451.05,A -85,B 0,C 180,E1 -29730.026,E2 -29730.026} C_VEL
LIN {X 0,Y 83.217,Z 463.197,A -85,B 0,C 180,E1 -29731.376,E2 -29731.376} C_VEL
LIN {X 0,Y 77.936,Z 475.099,A -85,B 0,C 180,E1 -29733.482,E2 -29733.482} C_VEL
LIN {X 0,Y 72.6,Z 484.73,A -85,B 0,C 180,E1 -29735.847,E2 -29735.847} C_VEL
LIN {X 0,Y 66.068,Z 494.608,A -85,B 0,C 180,E1 -29739.304,E2 -29739.304} C_VEL
LIN {X 0,Y 58.697,Z 503.948,A -85,B 0,C 180,E1 -29744.086,E2 -29744.086} C_VEL
LIN {X 0,Y 50.688,Z 512.858,A -85,B 0,C 180,E1 -29751.404,E2 -29751.404} C_VEL
LIN {X 0,Y 43.683,Z 519.995,A -85,B 0,C 180,E1 -29761.149,E2 -29761.149} C_VEL
LIN {X 0,Y 38.219,Z 525.69,A -85,B 0,C 180,E1 -29773.997,E2 -29773.997} C_VEL
LIN {X 0,Y 34.751,Z 530.198,A -85,B 0,C 180,E1 -29790.008,E2 -29790.008} C_VEL
LIN {X 0,Y 33.87,Z 532.599,A -85,B 0,C 180,E1 -29801.984,E2 -29801.984} C_VEL
LIN {X 0,Y 34.344,Z 534.568,A -85,B 0,C 180,E1 -29814.168,E2 -29814.168} C_VEL
LIN {X 0,Y 38.308,Z 536.851,A -85,B 0,C 180,E1 -29832.789,E2 -29832.789} C_VEL
LIN {X 0,Y 43.336,Z 537.772,A -85,B 0,C 180,E1 -29844.191,E2 -29844.191} C_VEL
LIN {X 0,Y 48.145,Z 538.006,A -85,B 0,C 180,E1 -29851.158,E2 -29851.158} C_VEL
LIN {X 0,Y 53.511,Z 537.791,A -85,B 0,C 180,E1 -29856.845,E2 -29856.845} C_VEL
LIN {X 0,Y 59.28,Z 537.172,A -85,B 0,C 180,E1 -29861.537,E2 -29861.537} C_VEL
LIN {X 0,Y 65.364,Z 536.143,A -85,B 0,C 180,E1 -29865.41,E2 -29865.41} C_VEL
LIN {X 0,Y 72.103,Z 534.519,A -85,B 0,C 180,E1 -29868.758,E2 -29868.758} C_VEL
LIN {X 0,Y 81.543,Z 531.518,A -85,B 0,C 180,E1 -29872.398,E2 -29872.398} C_VEL
LIN {X 0,Y 92.425,Z 526.901,A -85,B 0,C 180,E1 -29875.639,E2 -29875.639} C_VEL
LIN {X 0,Y 103.72,Z 520.73,A -85,B 0,C 180,E1 -29878.168,E2 -29878.168} C_VEL
LIN {X 0,Y 113.901,Z 513.725,A -85,B 0,C 180,E1 -29880,E2 -29880} C_VEL
LIN {X 0,Y 123.027,Z 506.034,A -85,B 0,C 180,E1 -29881.347,E2 -29881.347} C_VEL
LIN {X 0,Y 132.794,Z 495.934,A -85,B 0,C 180,E1 -29882.603,E2 -29882.603} C_VEL
LIN {X 0,Y 140.831,Z 485.605,A -85,B 0,C 180,E1 -29883.536,E2 -29883.536} C_VEL
LIN {X 0,Y 148.007,Z 474.001,A -85,B 0,C 180,E1 -29884.296,E2 -29884.296} C_VEL
LIN {X 0,Y 151.561,Z 467.064,A -85,B 0,C 180,E1 -29884.654,E2 -29884.654} C_VEL
LIN {X 0,Y 151.95,Z 466.146,A -85,B 0,C 180,E1 -29885.308,E2 -29885.308} C_VEL
LIN {X 0,Y 151.917,Z 466.472,A -85,B 0,C 180,E1 -29888.327,E2 -29888.327} C_VEL
LIN {X 0,Y 151.287,Z 467.896,A -85,B 0,C 180,E1 -29888.701,E2 -29888.701} C_VEL
LIN {X 0,Y 144.933,Z 479.629,A -85,B 0,C 180,E1 -29889.153,E2 -29889.153} C_VEL
LIN {X 0,Y 137.276,Z 490.853,A -85,B 0,C 180,E1 -29889.752,E2 -29889.752} C_VEL
LIN {X 0,Y 128.67,Z 500.944,A -85,B 0,C 180,E1 -29890.52,E2 -29890.52} C_VEL
LIN {X 0,Y 120.15,Z 509.19,A -85,B 0,C 180,E1 -29891.537,E2 -29891.537} C_VEL
LIN {X 0,Y 109.989,Z 517.29,A -85,B 0,C 180,E1 -29892.976,E2 -29892.976} C_VEL
LIN {X 0,Y 101.573,Z 522.828,A -85,B 0,C 180,E1 -29894.369,E2 -29894.369} C_VEL
LIN {X 0,Y 91.608,Z 528.265,A -85,B 0,C 180,E1 -29896.459,E2 -29896.459} C_VEL
LIN {X 0,Y 81.825,Z 532.546,A -85,B 0,C 180,E1 -29899.119,E2 -29899.119} C_VEL
LIN {X 0,Y 70.27,Z 536.408,A -85,B 0,C 180,E1 -29903.581,E2 -29903.581} C_VEL
LIN {X 0,Y 63.208,Z 538.101,A -85,B 0,C 180,E1 -29907.18,E2 -29907.18} C_VEL
LIN {X 0,Y 51.88,Z 539.782,A -85,B 0,C 180,E1 -29915.621,E2 -29915.621} C_VEL
LIN {X 0,Y 46.801,Z 540.06,A -85,B 0,C 180,E1 -29921.328,E2 -29921.328} C_VEL
LIN {X 0,Y 38.739,Z 539.414,A -85,B 0,C 180,E1 -29937.018,E2 -29937.018} C_VEL
LIN {X 0,Y 34.727,Z 537.251,A -85,B 0,C 180,E1 -29958.315,E2 -29958.315} C_VEL
LIN {X 0,Y 34.429,Z 535.529,A -85,B 0,C 180,E1 -29969.992,E2 -29969.992} C_VEL
LIN {X 0,Y 35.186,Z 532.003,A -85,B 0,C 180,E1 -29987.425,E2 -29987.425} C_VEL
LIN {X 0,Y 38.533,Z 527.317,A -85,B 0,C 180,E1 -30003.164,E2 -30003.164} C_VEL
LIN {X 0,Y 45.355,Z 520.231,A -85,B 0,C 180,E1 -30017.385,E2 -30017.385} C_VEL
LIN {X 0,Y 52.536,Z 512.664,A -85,B 0,C 180,E1 -30026.331,E2 -30026.331} C_VEL
LIN {X 0,Y 56.72,Z 507.903,A -85,B 0,C 180,E1 -30030.14,E2 -30030.14} C_VEL
LIN {X 0,Y 62.539,Z 500.977,A -85,B 0,C 180,E1 -30034.019,E2 -30034.019} C_VEL
LIN {X 0,Y 69.321,Z 491.605,A -85,B 0,C 180,E1 -30037.673,E2 -30037.673} C_VEL
LIN {X 0,Y 75.498,Z 481.356,A -85,B 0,C 180,E1 -30040.465,E2 -30040.465} C_VEL
LIN {X 0,Y 80.281,Z 471.992,A -85,B 0,C 180,E1 -30042.166,E2 -30042.166} C_VEL
LIN {X 0,Y 85.523,Z 458.954,A -85,B 0,C 180,E1 -30043.814,E2 -30043.814} C_VEL
LIN {X 0,Y 89.221,Z 446.383,A -85,B 0,C 180,E1 -30044.825,E2 -30044.825} C_VEL
LIN {X 0,Y 91.744,Z 432.705,A -85,B 0,C 180,E1 -30045.526,E2 -30045.526} C_VEL
LIN {X 0,Y 94.009,Z 412.345,A -85,B 0,C 180,E1 -30046.343,E2 -30046.343} C_VEL
LIN {X 0,Y 92.456,Z 407.562,A -85,B 0,C 180,E1 -30050.28,E2 -30050.28} C_VEL
LIN {X 0,Y 90.943,Z 403.247,A -85,B 0,C 180,E1 -30055.341,E2 -30055.341} C_VEL
LIN {X 0,Y 89.947,Z 399.752,A -85,B 0,C 180,E1 -30061.17,E2 -30061.17} C_VEL
LIN {X 0,Y 89.591,Z 399.458,A -85,B 0,C 180,E1 -30064.499,E2 -30064.499} C_VEL
LIN {X 0,Y 89.795,Z 400.083,A -85,B 0,C 180,E1 -30072.688,E2 -30072.688} C_VEL
LIN {X 0,Y 91.083,Z 404.05,A -85,B 0,C 180,E1 -30079.969,E2 -30079.969} C_VEL
LIN {X 0,Y 92.48,Z 407.707,A -85,B 0,C 180,E1 -30084.415,E2 -30084.415} C_VEL
LIN {X 0,Y 93.915,Z 412.083,A -85,B 0,C 180,E1 -30088.059,E2 -30088.059} C_VEL
LIN {X 0,Y 92.445,Z 425.803,A -85,B 0,C 180,E1 -30088.64,E2 -30088.64} C_VEL
LIN {X 0,Y 91.472,Z 431.639,A -85,B 0,C 180,E1 -30088.45,E2 -30088.45} C_VEL
LIN {X 0,Y 88.788,Z 441.002,A -85,B 0,C 180,E1 -30087.152,E2 -30087.152} C_VEL
LIN {X 0,Y 85.504,Z 450.192,A -85,B 0,C 180,E1 -30085.917,E2 -30085.917} C_VEL
LIN {X 0,Y 83.49,Z 455.753,A -85,B 0,C 180,E1 -30085.948,E2 -30085.948} C_VEL
LIN {X 0,Y 79.046,Z 467.08,A -85,B 0,C 180,E1 -30087.248,E2 -30087.248} C_VEL
LIN {X 0,Y 73.485,Z 478.282,A -85,B 0,C 180,E1 -30089.236,E2 -30089.236} C_VEL
LIN {X 0,Y 67.656,Z 487.772,A -85,B 0,C 180,E1 -30091.487,E2 -30091.487} C_VEL
LIN {X 0,Y 60.085,Z 498.033,A -85,B 0,C 180,E1 -30095.047,E2 -30095.047} C_VEL
LIN {X 0,Y 52.487,Z 506.668,A -85,B 0,C 180,E1 -30099.663,E2 -30099.663} C_VEL
LIN {X 0,Y 43.965,Z 515.042,A -85,B 0,C 180,E1 -30107.214,E2 -30107.214} C_VEL
LIN {X 0,Y 36.446,Z 521.793,A -85,B 0,C 180,E1 -30117.984,E2 -30117.984} C_VEL
LIN {X 0,Y 29.807,Z 527.986,A -85,B 0,C 180,E1 -30136.373,E2 -30136.373} C_VEL
LIN {X 0,Y 26.925,Z 532.04,A -85,B 0,C 180,E1 -30157.51,E2 -30157.51} C_VEL
LIN {X 0,Y 27.817,Z 535.046,A -85,B 0,C 180,E1 -30180.363,E2 -30180.363} C_VEL
LIN {X 0,Y 32.54,Z 537.078,A -85,B 0,C 180,E1 -30199.612,E2 -30199.612} C_VEL
LIN {X 0,Y 39.465,Z 538.107,A -85,B 0,C 180,E1 -30212.939,E2 -30212.939} C_VEL
LIN {X 0,Y 49.787,Z 538.096,A -85,B 0,C 180,E1 -30223.601,E2 -30223.601} C_VEL
LIN {X 0,Y 57.359,Z 537.343,A -85,B 0,C 180,E1 -30228.604,E2 -30228.604} C_VEL
LIN {X 0,Y 63.897,Z 536.24,A -85,B 0,C 180,E1 -30231.878,E2 -30231.878} C_VEL
LIN {X 0,Y 74.016,Z 533.742,A -85,B 0,C 180,E1 -30235.604,E2 -30235.604} C_VEL
LIN {X 0,Y 84.369,Z 530.168,A -85,B 0,C 180,E1 -30238.501,E2 -30238.501} C_VEL
LIN {X 0,Y 94.89,Z 525.405,A -85,B 0,C 180,E1 -30240.776,E2 -30240.776} C_VEL
LIN {X 0,Y 105.525,Z 519.309,A -85,B 0,C 180,E1 -30242.517,E2 -30242.517} C_VEL
LIN {X 0,Y 115.882,Z 511.933,A -85,B 0,C 180,E1 -30243.899,E2 -30243.899} C_VEL
LIN {X 0,Y 125.219,Z 503.777,A -85,B 0,C 180,E1 -30244.957,E2 -30244.957} C_VEL
LIN {X 0,Y 134.231,Z 494.071,A -85,B 0,C 180,E1 -30245.837,E2 -30245.837} C_VEL
LIN {X 0,Y 141.479,Z 484.522,A -85,B 0,C 180,E1 -30246.523,E2 -30246.523} C_VEL
LIN {X 0,Y 133.653,Z 494.848,A -85,B 0,C 180,E1 -30247.001,E2 -30247.001} C_VEL
LIN {X 0,Y 125.857,Z 503.299,A -85,B 0,C 180,E1 -30247.604,E2 -30247.604} C_VEL
LIN {X 0,Y 118.936,Z 509.64,A -85,B 0,C 180,E1 -30248.193,E2 -30248.193} C_VEL
LIN {X 0,Y 108.617,Z 517.619,A -85,B 0,C 180,E1 -30249.33,E2 -30249.33} C_VEL
LIN {X 0,Y 100.051,Z 523.049,A -85,B 0,C 180,E1 -30250.436,E2 -30250.436} C_VEL
LIN {X 0,Y 89.852,Z 528.39,A -85,B 0,C 180,E1 -30252.107,E2 -30252.107} C_VEL
LIN {X 0,Y 79.783,Z 532.581,A -85,B 0,C 180,E1 -30254.296,E2 -30254.296} C_VEL
LIN {X 0,Y 73.174,Z 534.822,A -85,B 0,C 180,E1 -30256.155,E2 -30256.155} C_VEL
LIN {X 0,Y 66.677,Z 536.6,A -85,B 0,C 180,E1 -30258.434,E2 -30258.434} C_VEL
LIN {X 0,Y 54.054,Z 538.96,A -85,B 0,C 180,E1 -30264.467,E2 -30264.467} C_VEL
LIN {X 0,Y 48.076,Z 539.575,A -85,B 0,C 180,E1 -30268.693,E2 -30268.693} C_VEL
LIN {X 0,Y 37.303,Z 539.602,A -85,B 0,C 180,E1 -30281.085,E2 -30281.085} C_VEL
LIN {X 0,Y 29.698,Z 538.124,A -85,B 0,C 180,E1 -30301.74,E2 -30301.74} C_VEL
LIN {X 0,Y 27.813,Z 536.802,A -85,B 0,C 180,E1 -30315.353,E2 -30315.353} C_VEL
LIN {X 0,Y 27.345,Z 535.009,A -85,B 0,C 180,E1 -30329.989,E2 -30329.989} C_VEL
LIN {X 0,Y 28.455,Z 531.391,A -85,B 0,C 180,E1 -30351.734,E2 -30351.734} C_VEL
LIN {X 0,Y 32.784,Z 526.611,A -85,B 0,C 180,E1 -30370.012,E2 -30370.012} C_VEL
LIN {X 0,Y 40.842,Z 519.421,A -85,B 0,C 180,E1 -30384.808,E2 -30384.808} C_VEL
LIN {X 0,Y 48.768,Z 511.816,A -85,B 0,C 180,E1 -30393.305,E2 -30393.305} C_VEL
LIN {X 0,Y 54.172,Z 506.192,A -85,B 0,C 180,E1 -30397.095,E2 -30397.095} C_VEL
LIN {X 0,Y 62.083,Z 496.791,A -85,B 0,C 180,E1 -30401.438,E2 -30401.438} C_VEL
LIN {X 0,Y 68.513,Z 487.795,A -85,B 0,C 180,E1 -30404.068,E2 -30404.068} C_VEL
LIN {X 0,Y 75.1,Z 476.738,A -85,B 0,C 180,E1 -30406.126,E2 -30406.126} C_VEL
LIN {X 0,Y 80.879,Z 464.247,A -85,B 0,C 180,E1 -30407.82,E2 -30407.82} C_VEL
LIN {X 0,Y 85.06,Z 452.408,A -85,B 0,C 180,E1 -30408.84,E2 -30408.84} C_VEL
LIN {X 0,Y 88.2,Z 439.71,A -85,B 0,C 180,E1 -30409.508,E2 -30409.508} C_VEL
LIN {X 0,Y 90.46,Z 423.67,A -85,B 0,C 180,E1 -30410.067,E2 -30410.067} C_VEL
LIN {X 0,Y 91.313,Z 415.651,A -85,B 0,C 180,E1 -30410.466,E2 -30410.466} C_VEL
LIN {X 0,Y 90.015,Z 411.156,A -85,B 0,C 180,E1 -30415.101,E2 -30415.101} C_VEL
LIN {X 0,Y 89.242,Z 408.428,A -85,B 0,C 180,E1 -30419.154,E2 -30419.154} C_VEL
LIN {X 0,Y 88.917,Z 406.681,A -85,B 0,C 180,E1 -30422.265,E2 -30422.265} C_VEL
LIN {X 0,Y 88.64,Z 406.676,A -85,B 0,C 180,E1 -30429.124,E2 -30429.124} C_VEL
LIN {X 0,Y 88.863,Z 407.284,A -85,B 0,C 180,E1 -30432.468,E2 -30432.468} C_VEL
LIN {X 0,Y 89.735,Z 410.573,A -85,B 0,C 180,E1 -30438.383,E2 -30438.383} C_VEL
LIN {X 0,Y 90.811,Z 413.984,A -85,B 0,C 180,E1 -30442.549,E2 -30442.549} C_VEL
LIN {X 0,Y 91.255,Z 415.583,A -85,B 0,C 180,E1 -30444,E2 -30444} C_VEL
LIN {X 0,Y 89.56,Z 430.207,A -85,B 0,C 180,E1 -30444.542,E2 -30444.542} C_VEL
LIN {X 0,Y 87.124,Z 443.463,A -85,B 0,C 180,E1 -30445.199,E2 -30445.199} C_VEL
LIN {X 0,Y 83.49,Z 455.753,A -85,B 0,C 180,E1 -30445.948,E2 -30445.948} C_VEL
LIN {X 0,Y 81.281,Z 461.264,A -85,B 0,C 180,E1 -30446.091,E2 -30446.091} C_VEL
LIN {X 0,Y 74.646,Z 473.326,A -85,B 0,C 180,E1 -30444.854,E2 -30444.854} C_VEL
LIN {X 0,Y 70.403,Z 479.973,A -85,B 0,C 180,E1 -30444.465,E2 -30444.465} C_VEL
LIN {X 0,Y 68.268,Z 483.249,A -85,B 0,C 180,E1 -30444.775,E2 -30444.775} C_VEL
LIN {X 0,Y 61.375,Z 493.058,A -85,B 0,C 180,E1 -30447.097,E2 -30447.097} C_VEL
LIN {X 0,Y 53.055,Z 502.842,A -85,B 0,C 180,E1 -30450.58,E2 -30450.58} C_VEL
LIN {X 0,Y 43.555,Z 512.038,A -85,B 0,C 180,E1 -30456.228,E2 -30456.228} C_VEL
LIN {X 0,Y 34.661,Z 519.443,A -85,B 0,C 180,E1 -30464.805,E2 -30464.805} C_VEL
LIN {X 0,Y 26.904,Z 525.382,A -85,B 0,C 180,E1 -30478.516,E2 -30478.516} C_VEL
LIN {X 0,Y 21.431,Z 529.953,A -85,B 0,C 180,E1 -30499.689,E2 -30499.689} C_VEL
LIN {X 0,Y 19.777,Z 533.7,A -85,B 0,C 180,E1 -30530.831,E2 -30530.831} C_VEL
LIN {X 0,Y 21.818,Z 535.508,A -85,B 0,C 180,E1 -30550.124,E2 -30550.124} C_VEL
LIN {X 0,Y 27.403,Z 537.299,A -85,B 0,C 180,E1 -30569.139,E2 -30569.139} C_VEL
LIN {X 0,Y 36.69,Z 538.414,A -85,B 0,C 180,E1 -30583.309,E2 -30583.309} C_VEL
LIN {X 0,Y 47.015,Z 538.39,A -85,B 0,C 180,E1 -30591.403,E2 -30591.403} C_VEL
LIN {X 0,Y 56.363,Z 537.507,A -85,B 0,C 180,E1 -30596.032,E2 -30596.032} C_VEL
LIN {X 0,Y 68.345,Z 535.206,A -85,B 0,C 180,E1 -30600,E2 -30600} C_VEL
LIN {X 0,Y 80.927,Z 531.412,A -85,B 0,C 180,E1 -30602.866,E2 -30602.866} C_VEL
LIN {X 0,Y 91.678,Z 526.968,A -85,B 0,C 180,E1 -30604.715,E2 -30604.715} C_VEL
LIN {X 0,Y 98.881,Z 523.31,A -85,B 0,C 180,E1 -30605.681,E2 -30605.681} C_VEL
LIN {X 0,Y 99.014,Z 523.27,A -85,B 0,C 180,E1 -30606.405,E2 -30606.405} C_VEL
LIN {X 0,Y 89.662,Z 528.032,A -85,B 0,C 180,E1 -30607.483,E2 -30607.483} C_VEL
LIN {X 0,Y 78.33,Z 532.616,A -85,B 0,C 180,E1 -30609.246,E2 -30609.246} C_VEL
LIN {X 0,Y 71.519,Z 534.787,A -85,B 0,C 180,E1 -30610.662,E2 -30610.662} C_VEL
LIN {X 0,Y 58.097,Z 537.842,A -85,B 0,C 180,E1 -30614.57,E2 -30614.57} C_VEL
LIN {X 0,Y 45.088,Z 539.353,A -85,B 0,C 180,E1 -30620.717,E2 -30620.717} C_VEL
LIN {X 0,Y 33.059,Z 539.279,A -85,B 0,C 180,E1 -30631.733,E2 -30631.733} C_VEL
LIN {X 0,Y 23.667,Z 537.722,A -85,B 0,C 180,E1 -30653.55,E2 -30653.55} C_VEL
LIN {X 0,Y 21.032,Z 536.327,A -85,B 0,C 180,E1 -30670.464,E2 -30670.464} C_VEL
LIN {X 0,Y 20.242,Z 534.487,A -85,B 0,C 180,E1 -30689.986,E2 -30689.986} C_VEL
LIN {X 0,Y 21.997,Z 530.781,A -85,B 0,C 180,E1 -30718.621,E2 -30718.621} C_VEL
LIN {X 0,Y 27.685,Z 525.904,A -85,B 0,C 180,E1 -30739.585,E2 -30739.585} C_VEL
LIN {X 0,Y 35.735,Z 519.746,A -85,B 0,C 180,E1 -30752.234,E2 -30752.234} C_VEL
LIN {X 0,Y 44.743,Z 512.025,A -85,B 0,C 180,E1 -30760.444,E2 -30760.444} C_VEL
LIN {X 0,Y 50.773,Z 506.174,A -85,B 0,C 180,E1 -30763.929,E2 -30763.929} C_VEL
LIN {X 0,Y 57.704,Z 498.547,A -85,B 0,C 180,E1 -30766.97,E2 -30766.97} C_VEL
LIN {X 0,Y 65.229,Z 488.775,A -85,B 0,C 180,E1 -30769.44,E2 -30769.44} C_VEL
LIN {X 0,Y 72.003,Z 478.073,A -85,B 0,C 180,E1 -30771.184,E2 -30771.184} C_VEL
LIN {X 0,Y 77.971,Z 466.077,A -85,B 0,C 180,E1 -30772.488,E2 -30772.488} C_VEL
LIN {X 0,Y 82.844,Z 453.07,A -85,B 0,C 180,E1 -30773.42,E2 -30773.42} C_VEL
LIN {X 0,Y 86.097,Z 440.778,A -85,B 0,C 180,E1 -30773.953,E2 -30773.953} C_VEL
LIN {X 0,Y 88.474,Z 425.068,A -85,B 0,C 180,E1 -30774.414,E2 -30774.414} C_VEL
LIN {X 0,Y 89.1,Z 419.492,A -85,B 0,C 180,E1 -30774.662,E2 -30774.662} C_VEL
LIN {X 0,Y 88.227,Z 415.558,A -85,B 0,C 180,E1 -30779.715,E2 -30779.715} C_VEL
LIN {X 0,Y 87.911,Z 413.638,A -85,B 0,C 180,E1 -30783.438,E2 -30783.438} C_VEL
LIN {X 0,Y 87.846,Z 413.937,A -85,B 0,C 180,E1 -30790.811,E2 -30790.811} C_VEL
LIN {X 0,Y 88.444,Z 417.064,A -85,B 0,C 180,E1 -30796.68,E2 -30796.68} C_VEL
LIN {X 0,Y 89.068,Z 419.448,A -85,B 0,C 180,E1 -30799.828,E2 -30799.828} C_VEL
LIN {X 0,Y 86.683,Z 436.744,A -85,B 0,C 180,E1 -30800.301,E2 -30800.301} C_VEL
LIN {X 0,Y 83.7,Z 449.236,A -85,B 0,C 180,E1 -30800.881,E2 -30800.881} C_VEL
